gfCNCPoint2[25191] = {X 190.9402, Y 34.0721, Z -3.8333, A 0.000, B 0.000, C 0.000 }
gfCNCPoint2[25192] = {X 189.2026, Y 34.2446, Z -3.8333, A 0.000, B 0.000, C 0.000 }
gfCNCPoint2[25193] = {X 186.9380, Y 34.3837, Z -3.8333, A 0.000, B 0.000, C 0.000 }
gfCNCPoint2[25194] = {X 182.9821, Y 34.9758, Z -3.8333, A 0.000, B 0.000, C 0.000 }
gfCNCPoint2[25195] = {X 182.9821, Y 34.9758, Z -0.8333, A 0.000, B 0.000, C 0.000 }
gfCNCPoint2[25196] = {X 182.9821, Y 34.9758, Z 11.0000, A 0.000, B 0.000, C 0.000 }
gfCNCPoint2[25197] = {X 188.4961, Y 19.4662, Z 11.0000, A 0.000, B 0.000, C 0.000 }
gfCNCPoint2[25198] = {X 188.4961, Y 19.4662, Z 0.0000, A 0.000, B 0.000, C 0.000 }
gfCNCPoint2[25199] = {X 188.3884, Y 19.4281, Z -0.0306, A 0.000, B 0.000, C 0.000 }
gfCNCPoint2[25200] = {X 187.7714, Y 19.3596, Z -0.1969, A 0.000, B 0.000, C 0.000 }
gfCNCPoint2[25201] = {X 186.9109, Y 19.2596, Z -0.4291, A 0.000, B 0.000, C 0.000 }
gfCNCPoint2[25202] = {X 184.5930, Y 19.3671, Z -1.0508, A 0.000, B 0.000, C 0.000 }
gfCNCPoint2[25203] = {X 183.7430, Y 19.5468, Z -1.2836, A 0.000, B 0.000, C 0.000 }
gfCNCPoint2[25204] = {X 183.0416, Y 19.6905, Z -1.4754, A 0.000, B 0.000, C 0.000 }
gfCNCPoint2[25205] = {X 182.0251, Y 20.0604, Z -1.7653, A 0.000, B 0.000, C 0.000 }
gfCNCPoint2[25206] = {X 181.3955, Y 20.4012, Z -1.9571, A 0.000, B 0.000, C 0.000 }
gfCNCPoint2[25207] = {X 181.3396, Y 20.9128, Z -2.0950, A 0.000, B 0.000, C 0.000 }
gfCNCPoint2[25208] = {X 180.8645, Y 22.1268, Z -2.4443, A 0.000, B 0.000, C 0.000 }
gfCNCPoint2[25209] = {X 180.5584, Y 22.5405, Z -2.5822, A 0.000, B 0.000, C 0.000 }
gfCNCPoint2[25210] = {X 182.2910, Y 22.3346, Z -3.0498, A 0.000, B 0.000, C 0.000 }
gfCNCPoint2[25211] = {X 182.5945, Y 22.3099, Z -3.1314, A 0.000, B 0.000, C 0.000 }
gfCNCPoint2[25212] = {X 184.3413, Y 22.2338, Z -3.5999, A 0.000, B 0.000, C 0.000 }
gfCNCPoint2[25213] = {X 184.7767, Y 22.2187, Z -3.7166, A 0.000, B 0.000, C 0.000 }
gfCNCPoint2[25214] = {X 185.2120, Y 22.2003, Z -3.8333, A 0.000, B 0.000, C 0.000 }
gfCNCPoint2[25215] = {X 187.5425, Y 22.0778, Z -3.8333, A 0.000, B 0.000, C 0.000 }
gfCNCPoint2[25216] = {X 189.8700, Y 21.9074, Z -3.8333, A 0.000, B 0.000, C 0.000 }
gfCNCPoint2[25217] = {X 190.4716, Y 21.8313, Z -3.8333, A 0.000, B 0.000, C 0.000 }
gfCNCPoint2[25218] = {X 191.0588, Y 21.6799, Z -3.8333, A 0.000, B 0.000, C 0.000 }
gfCNCPoint2[25219] = {X 191.0686, Y 21.1639, Z -3.8333, A 0.000, B 0.000, C 0.000 }
gfCNCPoint2[25220] = {X 190.8728, Y 20.6864, Z -3.8333, A 0.000, B 0.000, C 0.000 }
gfCNCPoint2[25221] = {X 190.5036, Y 20.3258, Z -3.8333, A 0.000, B 0.000, C 0.000 }
gfCNCPoint2[25222] = {X 189.6459, Y 19.8651, Z -3.8333, A 0.000, B 0.000, C 0.000 }
gfCNCPoint2[25223] = {X 188.7281, Y 19.5404, Z -3.8333, A 0.000, B 0.000, C 0.000 }
gfCNCPoint2[25224] = {X 187.7714, Y 19.3596, Z -3.8333, A 0.000, B 0.000, C 0.000 }
gfCNCPoint2[25225] = {X 186.4245, Y 19.2765, Z -3.8333, A 0.000, B 0.000, C 0.000 }
gfCNCPoint2[25226] = {X 185.0764, Y 19.3391, Z -3.8333, A 0.000, B 0.000, C 0.000 }
gfCNCPoint2[25227] = {X 183.7430, Y 19.5468, Z -3.8333, A 0.000, B 0.000, C 0.000 }
gfCNCPoint2[25228] = {X 182.5378, Y 19.8876, Z -3.8333, A 0.000, B 0.000, C 0.000 }
gfCNCPoint2[25229] = {X 181.3955, Y 20.4012, Z -3.8333, A 0.000, B 0.000, C 0.000 }
gfCNCPoint2[25230] = {X 181.2441, Y 21.1600, Z -3.8333, A 0.000, B 0.000, C 0.000 }
gfCNCPoint2[25231] = {X 180.9622, Y 21.8805, Z -3.8333, A 0.000, B 0.000, C 0.000 }
gfCNCPoint2[25232] = {X 180.5584, Y 22.5405, Z -3.8333, A 0.000, B 0.000, C 0.000 }
gfCNCPoint2[25233] = {X 182.4470, Y 22.3518, Z -3.8333, A 0.000, B 0.000, C 0.000 }
gfCNCPoint2[25234] = {X 184.3413, Y 22.2338, Z -3.8333, A 0.000, B 0.000, C 0.000 }
gfCNCPoint2[25235] = {X 184.7767, Y 22.2179, Z -3.8333, A 0.000, B 0.000, C 0.000 }
gfCNCPoint2[25236] = {X 185.2120, Y 22.2003, Z -3.8333, A 0.000, B 0.000, C 0.000 }
gfCNCPoint2[25237] = {X 181.2194, Y 22.1003, Z -3.8333, A 0.000, B 0.000, C 0.000 }
gfCNCPoint2[25238] = {X 185.2154, Y 22.2803, Z -3.8333, A 0.000, B 0.000, C 0.000 }
gfCNCPoint2[25239] = {X 187.5451, Y 22.1578, Z -3.8333, A 0.000, B 0.000, C 0.000 }
gfCNCPoint2[25240] = {X 189.8718, Y 21.9874, Z -3.8333, A 0.000, B 0.000, C 0.000 }
gfCNCPoint2[25241] = {X 190.5070, Y 21.9059, Z -3.8333, A 0.000, B 0.000, C 0.000 }
gfCNCPoint2[25242] = {X 191.1260, Y 21.7420, Z -3.8333, A 0.000, B 0.000, C 0.000 }
gfCNCPoint2[25243] = {X 191.1525, Y 21.1792, Z -3.8333, A 0.000, B 0.000, C 0.000 }
gfCNCPoint2[25244] = {X 190.9475, Y 20.6544, Z -3.8333, A 0.000, B 0.000, C 0.000 }
gfCNCPoint2[25245] = {X 190.5467, Y 20.2585, Z -3.8333, A 0.000, B 0.000, C 0.000 }
gfCNCPoint2[25246] = {X 189.6789, Y 19.7922, Z -3.8333, A 0.000, B 0.000, C 0.000 }
gfCNCPoint2[25247] = {X 188.7502, Y 19.4636, Z -3.8333, A 0.000, B 0.000, C 0.000 }
gfCNCPoint2[25248] = {X 187.7823, Y 19.2803, Z -3.8333, A 0.000, B 0.000, C 0.000 }
gfCNCPoint2[25249] = {X 186.4270, Y 19.1965, Z -3.8333, A 0.000, B 0.000, C 0.000 }
gfCNCPoint2[25250] = {X 185.0706, Y 19.2593, Z -3.8333, A 0.000, B 0.000, C 0.000 }
gfCNCPoint2[25251] = {X 183.7289, Y 19.4680, Z -3.8333, A 0.000, B 0.000, C 0.000 }
gfCNCPoint2[25252] = {X 182.4922, Y 19.8190, Z -3.8333, A 0.000, B 0.000, C 0.000 }
gfCNCPoint2[25253] = {X 181.3215, Y 20.3504, Z -3.8333, A 0.000, B 0.000, C 0.000 }
gfCNCPoint2[25254] = {X 181.1595, Y 21.1706, Z -3.8333, A 0.000, B 0.000, C 0.000 }
gfCNCPoint2[25255] = {X 180.8425, Y 21.9443, Z -3.8333, A 0.000, B 0.000, C 0.000 }
gfCNCPoint2[25256] = {X 180.3824, Y 22.6424, Z -3.8333, A 0.000, B 0.000, C 0.000 }
gfCNCPoint2[25257] = {X 182.3593, Y 22.4392, Z -3.8333, A 0.000, B 0.000, C 0.000 }
gfCNCPoint2[25258] = {X 184.3427, Y 22.3138, Z -3.8333, A 0.000, B 0.000, C 0.000 }
gfCNCPoint2[25259] = {X 184.7791, Y 22.2979, Z -3.8333, A 0.000, B 0.000, C 0.000 }
gfCNCPoint2[25260] = {X 185.2154, Y 22.2803, Z -3.8333, A 0.000, B 0.000, C 0.000 }
gfCNCPoint2[25261] = {X 189.1819, Y 21.7636, Z -3.8333, A 0.000, B 0.000, C 0.000 }
gfCNCPoint2[25262] = {X 181.2228, Y 22.1802, Z -3.8333, A 0.000, B 0.000, C 0.000 }
gfCNCPoint2[25263] = {X 185.2187, Y 22.3602, Z -3.8333, A 0.000, B 0.000, C 0.000 }
gfCNCPoint2[25264] = {X 187.5497, Y 22.2376, Z -3.8333, A 0.000, B 0.000, C 0.000 }
gfCNCPoint2[25265] = {X 189.8776, Y 22.0672, Z -3.8333, A 0.000, B 0.000, C 0.000 }
gfCNCPoint2[25266] = {X 190.5436, Y 21.9802, Z -3.8333, A 0.000, B 0.000, C 0.000 }
gfCNCPoint2[25267] = {X 191.1918, Y 21.8041, Z -3.8333, A 0.000, B 0.000, C 0.000 }
gfCNCPoint2[25268] = {X 191.2495, Y 21.3480, Z -3.8333, A 0.000, B 0.000, C 0.000 }
gfCNCPoint2[25269] = {X 191.1599, Y 20.8972, Z -3.8333, A 0.000, B 0.000, C 0.000 }
gfCNCPoint2[25270] = {X 190.9322, Y 20.4978, Z -3.8333, A 0.000, B 0.000, C 0.000 }
gfCNCPoint2[25271] = {X 190.5898, Y 20.1911, Z -3.8333, A 0.000, B 0.000, C 0.000 }
gfCNCPoint2[25272] = {X 189.7113, Y 19.7190, Z -3.8333, A 0.000, B 0.000, C 0.000 }
gfCNCPoint2[25273] = {X 188.7710, Y 19.3863, Z -3.8333, A 0.000, B 0.000, C 0.000 }
gfCNCPoint2[25274] = {X 187.7911, Y 19.2008, Z -3.8333, A 0.000, B 0.000, C 0.000 }
gfCNCPoint2[25275] = {X 186.4273, Y 19.1165, Z -3.8333, A 0.000, B 0.000, C 0.000 }
gfCNCPoint2[25276] = {X 185.0625, Y 19.1797, Z -3.8333, A 0.000, B 0.000, C 0.000 }
gfCNCPoint2[25277] = {X 183.7123, Y 19.3897, Z -3.8333, A 0.000, B 0.000, C 0.000 }
gfCNCPoint2[25278] = {X 182.4466, Y 19.7506, Z -3.8333, A 0.000, B 0.000, C 0.000 }
gfCNCPoint2[25279] = {X 181.2499, Y 20.2985, Z -3.8333, A 0.000, B 0.000, C 0.000 }
gfCNCPoint2[25280] = {X 181.2398, Y 20.3524, Z -3.8333, A 0.000, B 0.000, C 0.000 }
gfCNCPoint2[25281] = {X 181.0601, Y 21.2185, Z -3.8333, A 0.000, B 0.000, C 0.000 }
gfCNCPoint2[25282] = {X 180.7046, Y 22.0285, Z -3.8333, A 0.000, B 0.000, C 0.000 }
gfCNCPoint2[25283] = {X 180.1888, Y 22.7471, Z -3.8333, A 0.000, B 0.000, C 0.000 }
gfCNCPoint2[25284] = {X 182.2636, Y 22.5276, Z -3.8333, A 0.000, B 0.000, C 0.000 }
gfCNCPoint2[25285] = {X 184.3458, Y 22.3938, Z -3.8333, A 0.000, B 0.000, C 0.000 }
gfCNCPoint2[25286] = {X 184.7823, Y 22.3778, Z -3.8333, A 0.000, B 0.000, C 0.000 }
gfCNCPoint2[25287] = {X 185.2187, Y 22.3602, Z -3.8333, A 0.000, B 0.000, C 0.000 }
gfCNCPoint2[25288] = {X 189.1852, Y 21.8435, Z -3.8333, A 0.000, B 0.000, C 0.000 }
gfCNCPoint2[25289] = {X 181.2262, Y 22.2602, Z -3.8333, A 0.000, B 0.000, C 0.000 }
gfCNCPoint2[25290] = {X 185.2221, Y 22.4401, Z -3.8333, A 0.000, B 0.000, C 0.000 }
gfCNCPoint2[25291] = {X 187.5543, Y 22.3175, Z -3.8333, A 0.000, B 0.000, C 0.000 }
gfCNCPoint2[25292] = {X 189.8834, Y 22.1470, Z -3.8333, A 0.000, B 0.000, C 0.000 }
gfCNCPoint2[25293] = {X 190.5796, Y 22.0546, Z -3.8333, A 0.000, B 0.000, C 0.000 }
gfCNCPoint2[25294] = {X 191.2562, Y 21.8662, Z -3.8333, A 0.000, B 0.000, C 0.000 }
gfCNCPoint2[25295] = {X 191.3302, Y 21.3762, Z -3.8333, A 0.000, B 0.000, C 0.000 }
gfCNCPoint2[25296] = {X 191.2419, Y 20.8886, Z -3.8333, A 0.000, B 0.000, C 0.000 }
gfCNCPoint2[25297] = {X 191.0009, Y 20.4557, Z -3.8333, A 0.000, B 0.000, C 0.000 }
gfCNCPoint2[25298] = {X 190.6330, Y 20.1237, Z -3.8333, A 0.000, B 0.000, C 0.000 }
gfCNCPoint2[25299] = {X 189.7437, Y 19.6459, Z -3.8333, A 0.000, B 0.000, C 0.000 }
gfCNCPoint2[25300] = {X 188.7919, Y 19.3091, Z -3.8333, A 0.000, B 0.000, C 0.000 }
gfCNCPoint2[25301] = {X 187.7999, Y 19.1213, Z -3.8333, A 0.000, B 0.000, C 0.000 }
gfCNCPoint2[25302] = {X 186.4277, Y 19.0365, Z -3.8333, A 0.000, B 0.000, C 0.000 }
gfCNCPoint2[25303] = {X 185.0543, Y 19.1001, Z -3.8333, A 0.000, B 0.000, C 0.000 }
gfCNCPoint2[25304] = {X 183.6958, Y 19.3115, Z -3.8333, A 0.000, B 0.000, C 0.000 }
gfCNCPoint2[25305] = {X 182.4009, Y 19.6822, Z -3.8333, A 0.000, B 0.000, C 0.000 }
gfCNCPoint2[25306] = {X 181.1781, Y 20.2468, Z -3.8333, A 0.000, B 0.000, C 0.000 }
gfCNCPoint2[25307] = {X 181.1605, Y 20.3410, Z -3.8333, A 0.000, B 0.000, C 0.000 }
gfCNCPoint2[25308] = {X 180.9651, Y 21.2476, Z -3.8333, A 0.000, B 0.000, C 0.000 }
gfCNCPoint2[25309] = {X 180.5736, Y 22.0884, Z -3.8333, A 0.000, B 0.000, C 0.000 }
gfCNCPoint2[25310] = {X 180.0056, Y 22.8216, Z -3.8333, A 0.000, B 0.000, C 0.000 }
gfCNCPoint2[25311] = {X 180.1926, Y 22.8273, Z -3.8333, A 0.000, B 0.000, C 0.000 }
gfCNCPoint2[25312] = {X 182.2671, Y 22.6075, Z -3.8333, A 0.000, B 0.000, C 0.000 }
gfCNCPoint2[25313] = {X 184.3489, Y 22.4737, Z -3.8333, A 0.000, B 0.000, C 0.000 }
gfCNCPoint2[25314] = {X 184.7856, Y 22.4577, Z -3.8333, A 0.000, B 0.000, C 0.000 }
gfCNCPoint2[25315] = {X 185.2221, Y 22.4401, Z -3.8333, A 0.000, B 0.000, C 0.000 }
gfCNCPoint2[25316] = {X 189.1886, Y 21.9235, Z -3.8333, A 0.000, B 0.000, C 0.000 }
gfCNCPoint2[25317] = {X 181.2296, Y 22.3401, Z -3.8333, A 0.000, B 0.000, C 0.000 }
gfCNCPoint2[25318] = {X 185.2255, Y 22.5201, Z -3.8333, A 0.000, B 0.000, C 0.000 }
gfCNCPoint2[25319] = {X 187.5589, Y 22.3974, Z -3.8333, A 0.000, B 0.000, C 0.000 }
gfCNCPoint2[25320] = {X 189.8892, Y 22.2268, Z -3.8333, A 0.000, B 0.000, C 0.000 }
gfCNCPoint2[25321] = {X 190.6151, Y 22.1289, Z -3.8333, A 0.000, B 0.000, C 0.000 }
gfCNCPoint2[25322] = {X 191.3196, Y 21.9285, Z -3.8333, A 0.000, B 0.000, C 0.000 }
gfCNCPoint2[25323] = {X 191.4103, Y 21.4048, Z -3.8333, A 0.000, B 0.000, C 0.000 }
gfCNCPoint2[25324] = {X 191.3238, Y 20.8804, Z -3.8333, A 0.000, B 0.000, C 0.000 }
gfCNCPoint2[25325] = {X 191.0696, Y 20.4136, Z -3.8333, A 0.000, B 0.000, C 0.000 }
gfCNCPoint2[25326] = {X 190.6761, Y 20.0564, Z -3.8333, A 0.000, B 0.000, C 0.000 }
gfCNCPoint2[25327] = {X 189.7760, Y 19.5727, Z -3.8333, A 0.000, B 0.000, C 0.000 }
gfCNCPoint2[25328] = {X 188.8127, Y 19.2318, Z -3.8333, A 0.000, B 0.000, C 0.000 }
gfCNCPoint2[25329] = {X 187.8088, Y 19.0418, Z -3.8333, A 0.000, B 0.000, C 0.000 }
gfCNCPoint2[25330] = {X 186.4280, Y 18.9565, Z -3.8333, A 0.000, B 0.000, C 0.000 }
gfCNCPoint2[25331] = {X 185.0462, Y 19.0205, Z -3.8333, A 0.000, B 0.000, C 0.000 }
gfCNCPoint2[25332] = {X 183.6792, Y 19.2332, Z -3.8333, A 0.000, B 0.000, C 0.000 }
gfCNCPoint2[25333] = {X 182.3552, Y 19.6138, Z -3.8333, A 0.000, B 0.000, C 0.000 }
gfCNCPoint2[25334] = {X 181.1064, Y 20.1954, Z -3.8333, A 0.000, B 0.000, C 0.000 }
gfCNCPoint2[25335] = {X 181.0813, Y 20.3296, Z -3.8333, A 0.000, B 0.000, C 0.000 }
gfCNCPoint2[25336] = {X 180.8699, Y 21.2784, Z -3.8333, A 0.000, B 0.000, C 0.000 }
gfCNCPoint2[25337] = {X 180.4400, Y 22.1503, Z -3.8333, A 0.000, B 0.000, C 0.000 }
gfCNCPoint2[25338] = {X 179.8161, Y 22.8958, Z -3.8333, A 0.000, B 0.000, C 0.000 }
gfCNCPoint2[25339] = {X 180.1964, Y 22.9074, Z -3.8333, A 0.000, B 0.000, C 0.000 }
gfCNCPoint2[25340] = {X 182.2706, Y 22.6875, Z -3.8333, A 0.000, B 0.000, C 0.000 }
gfCNCPoint2[25341] = {X 184.3521, Y 22.5536, Z -3.8333, A 0.000, B 0.000, C 0.000 }
gfCNCPoint2[25342] = {X 184.7888, Y 22.5377, Z -3.8333, A 0.000, B 0.000, C 0.000 }
gfCNCPoint2[25343] = {X 185.2255, Y 22.5201, Z -3.8333, A 0.000, B 0.000, C 0.000 }
gfCNCPoint2[25344] = {X 189.1920, Y 22.0034, Z -3.8333, A 0.000, B 0.000, C 0.000 }
gfCNCPoint2[25345] = {X 185.1538, Y 22.6031, Z -3.8333, A 0.000, B 0.000, C 0.000 }
gfCNCPoint2[25346] = {X 185.2289, Y 22.6000, Z -3.8333, A 0.000, B 0.000, C 0.000 }
gfCNCPoint2[25347] = {X 187.5635, Y 22.4772, Z -3.8333, A 0.000, B 0.000, C 0.000 }
gfCNCPoint2[25348] = {X 189.8950, Y 22.3066, Z -3.8333, A 0.000, B 0.000, C 0.000 }
gfCNCPoint2[25349] = {X 190.6501, Y 22.2033, Z -3.8333, A 0.000, B 0.000, C 0.000 }
gfCNCPoint2[25350] = {X 191.3820, Y 21.9907, Z -3.8333, A 0.000, B 0.000, C 0.000 }
gfCNCPoint2[25351] = {X 191.4900, Y 21.4336, Z -3.8333, A 0.000, B 0.000, C 0.000 }
gfCNCPoint2[25352] = {X 191.4055, Y 20.8724, Z -3.8333, A 0.000, B 0.000, C 0.000 }
gfCNCPoint2[25353] = {X 191.1384, Y 20.3716, Z -3.8333, A 0.000, B 0.000, C 0.000 }
gfCNCPoint2[25354] = {X 190.7193, Y 19.9890, Z -3.8333, A 0.000, B 0.000, C 0.000 }
gfCNCPoint2[25355] = {X 189.8084, Y 19.4995, Z -3.8333, A 0.000, B 0.000, C 0.000 }
gfCNCPoint2[25356] = {X 188.8336, Y 19.1546, Z -3.8333, A 0.000, B 0.000, C 0.000 }
gfCNCPoint2[25357] = {X 187.8176, Y 18.9622, Z -3.8333, A 0.000, B 0.000, C 0.000 }
gfCNCPoint2[25358] = {X 186.4284, Y 18.8765, Z -3.8333, A 0.000, B 0.000, C 0.000 }
gfCNCPoint2[25359] = {X 185.0380, Y 18.9410, Z -3.8333, A 0.000, B 0.000, C 0.000 }
gfCNCPoint2[25360] = {X 183.6627, Y 19.1549, Z -3.8333, A 0.000, B 0.000, C 0.000 }
gfCNCPoint2[25361] = {X 182.3095, Y 19.5455, Z -3.8333, A 0.000, B 0.000, C 0.000 }
gfCNCPoint2[25362] = {X 181.0346, Y 20.1441, Z -3.8333, A 0.000, B 0.000, C 0.000 }
gfCNCPoint2[25363] = {X 181.0020, Y 20.3183, Z -3.8333, A 0.000, B 0.000, C 0.000 }
gfCNCPoint2[25364] = {X 180.8538, Y 21.0695, Z -3.8333, A 0.000, B 0.000, C 0.000 }
gfCNCPoint2[25365] = {X 180.5651, Y 21.7787, Z -3.8333, A 0.000, B 0.000, C 0.000 }
gfCNCPoint2[25366] = {X 180.1466, Y 22.4199, Z -3.8333, A 0.000, B 0.000, C 0.000 }
gfCNCPoint2[25367] = {X 179.6136, Y 22.9696, Z -3.8333, A 0.000, B 0.000, C 0.000 }
gfCNCPoint2[25368] = {X 180.2003, Y 22.9876, Z -3.8333, A 0.000, B 0.000, C 0.000 }
gfCNCPoint2[25369] = {X 182.2741, Y 22.7675, Z -3.8333, A 0.000, B 0.000, C 0.000 }
gfCNCPoint2[25370] = {X 184.3552, Y 22.6336, Z -3.8333, A 0.000, B 0.000, C 0.000 }
gfCNCPoint2[25371] = {X 184.7921, Y 22.6176, Z -3.8333, A 0.000, B 0.000, C 0.000 }
gfCNCPoint2[25372] = {X 185.2289, Y 22.6000, Z -3.8333, A 0.000, B 0.000, C 0.000 }
gfCNCPoint2[25373] = {X 185.1444, Y 20.6018, Z -3.8333, A 0.000, B 0.000, C 0.000 }
gfCNCPoint2[25374] = {X 185.1444, Y 20.6018, Z -0.8333, A 0.000, B 0.000, C 0.000 }
gfCNCPoint2[25375] = {X 185.1444, Y 20.6018, Z 11.0000, A 0.000, B 0.000, C 0.000 }
gfCNCPoint2[25376] = {X 256.2436, Y 19.7807, Z 11.0000, A 0.000, B 0.000, C 0.000 }
gfCNCPoint2[25377] = {X 256.2436, Y 19.7807, Z 0.0000, A 0.000, B 0.000, C 0.000 }
gfCNCPoint2[25378] = {X 251.5292, Y 19.7807, Z -1.2632, A 0.000, B 0.000, C 0.000 }
gfCNCPoint2[25379] = {X 250.8345, Y 19.7916, Z -1.4494, A 0.000, B 0.000, C 0.000 }
gfCNCPoint2[25380] = {X 250.1809, Y 19.7930, Z -1.6245, A 0.000, B 0.000, C 0.000 }
gfCNCPoint2[25381] = {X 249.4954, Y 19.8914, Z -1.8101, A 0.000, B 0.000, C 0.000 }
gfCNCPoint2[25382] = {X 248.8452, Y 20.0797, Z -1.9915, A 0.000, B 0.000, C 0.000 }
gfCNCPoint2[25383] = {X 248.7082, Y 20.1110, Z -2.0291, A 0.000, B 0.000, C 0.000 }
gfCNCPoint2[25384] = {X 248.6540, Y 20.1618, Z -2.0490, A 0.000, B 0.000, C 0.000 }
gfCNCPoint2[25385] = {X 248.4750, Y 20.7647, Z -2.2175, A 0.000, B 0.000, C 0.000 }
gfCNCPoint2[25386] = {X 248.4449, Y 21.8677, Z -2.5132, A 0.000, B 0.000, C 0.000 }
gfCNCPoint2[25387] = {X 248.5581, Y 22.3427, Z -2.6441, A 0.000, B 0.000, C 0.000 }
gfCNCPoint2[25388] = {X 248.8730, Y 22.4374, Z -2.7322, A 0.000, B 0.000, C 0.000 }
gfCNCPoint2[25389] = {X 249.2007, Y 22.4646, Z -2.8203, A 0.000, B 0.000, C 0.000 }
gfCNCPoint2[25390] = {X 250.4401, Y 22.5675, Z -3.1535, A 0.000, B 0.000, C 0.000 }
gfCNCPoint2[25391] = {X 251.6873, Y 22.5560, Z -3.4877, A 0.000, B 0.000, C 0.000 }
gfCNCPoint2[25392] = {X 252.9772, Y 22.5560, Z -3.8333, A 0.000, B 0.000, C 0.000 }
gfCNCPoint2[25393] = {X 257.4115, Y 22.5560, Z -3.8333, A 0.000, B 0.000, C 0.000 }
gfCNCPoint2[25394] = {X 257.4115, Y 19.7807, Z -3.8333, A 0.000, B 0.000, C 0.000 }
gfCNCPoint2[25395] = {X 251.5292, Y 19.7807, Z -3.8333, A 0.000, B 0.000, C 0.000 }
gfCNCPoint2[25396] = {X 250.8345, Y 19.7916, Z -3.8333, A 0.000, B 0.000, C 0.000 }
gfCNCPoint2[25397] = {X 249.8296, Y 19.8649, Z -3.8333, A 0.000, B 0.000, C 0.000 }
gfCNCPoint2[25398] = {X 248.8452, Y 20.0797, Z -3.8333, A 0.000, B 0.000, C 0.000 }
gfCNCPoint2[25399] = {X 248.7002, Y 20.1568, Z -3.8333, A 0.000, B 0.000, C 0.000 }
gfCNCPoint2[25400] = {X 248.6140, Y 20.2965, Z -3.8333, A 0.000, B 0.000, C 0.000 }
gfCNCPoint2[25401] = {X 248.4760, Y 20.9719, Z -3.8333, A 0.000, B 0.000, C 0.000 }
gfCNCPoint2[25402] = {X 248.4572, Y 21.6609, Z -3.8333, A 0.000, B 0.000, C 0.000 }
gfCNCPoint2[25403] = {X 248.5581, Y 22.3427, Z -3.8333, A 0.000, B 0.000, C 0.000 }
gfCNCPoint2[25404] = {X 248.8762, Y 22.4205, Z -3.8333, A 0.000, B 0.000, C 0.000 }
gfCNCPoint2[25405] = {X 249.2007, Y 22.4646, Z -3.8333, A 0.000, B 0.000, C 0.000 }
gfCNCPoint2[25406] = {X 250.4430, Y 22.5389, Z -3.8333, A 0.000, B 0.000, C 0.000 }
gfCNCPoint2[25407] = {X 251.6873, Y 22.5560, Z -3.8333, A 0.000, B 0.000, C 0.000 }
gfCNCPoint2[25408] = {X 252.9772, Y 22.5560, Z -3.8333, A 0.000, B 0.000, C 0.000 }
gfCNCPoint2[25409] = {X 248.9925, Y 22.2874, Z -3.8333, A 0.000, B 0.000, C 0.000 }
gfCNCPoint2[25410] = {X 252.9772, Y 22.6360, Z -3.8333, A 0.000, B 0.000, C 0.000 }
gfCNCPoint2[25411] = {X 257.4915, Y 22.6360, Z -3.8333, A 0.000, B 0.000, C 0.000 }
gfCNCPoint2[25412] = {X 257.4915, Y 19.7007, Z -3.8333, A 0.000, B 0.000, C 0.000 }
gfCNCPoint2[25413] = {X 251.5286, Y 19.7007, Z -3.8333, A 0.000, B 0.000, C 0.000 }
gfCNCPoint2[25414] = {X 250.8365, Y 19.7116, Z -3.8333, A 0.000, B 0.000, C 0.000 }
gfCNCPoint2[25415] = {X 249.8259, Y 19.7850, Z -3.8333, A 0.000, B 0.000, C 0.000 }
gfCNCPoint2[25416] = {X 248.8356, Y 19.9999, Z -3.8333, A 0.000, B 0.000, C 0.000 }
gfCNCPoint2[25417] = {X 248.6486, Y 20.0956, Z -3.8333, A 0.000, B 0.000, C 0.000 }
gfCNCPoint2[25418] = {X 248.5373, Y 20.2738, Z -3.8333, A 0.000, B 0.000, C 0.000 }
gfCNCPoint2[25419] = {X 248.3948, Y 20.9779, Z -3.8333, A 0.000, B 0.000, C 0.000 }
gfCNCPoint2[25420] = {X 248.3793, Y 21.6962, Z -3.8333, A 0.000, B 0.000, C 0.000 }
gfCNCPoint2[25421] = {X 248.4912, Y 22.4058, Z -3.8333, A 0.000, B 0.000, C 0.000 }
gfCNCPoint2[25422] = {X 248.8388, Y 22.4947, Z -3.8333, A 0.000, B 0.000, C 0.000 }
gfCNCPoint2[25423] = {X 249.1941, Y 22.5443, Z -3.8333, A 0.000, B 0.000, C 0.000 }
gfCNCPoint2[25424] = {X 250.4389, Y 22.6188, Z -3.8333, A 0.000, B 0.000, C 0.000 }
gfCNCPoint2[25425] = {X 251.6859, Y 22.6360, Z -3.8333, A 0.000, B 0.000, C 0.000 }
gfCNCPoint2[25426] = {X 252.9772, Y 22.6360, Z -3.8333, A 0.000, B 0.000, C 0.000 }
gfCNCPoint2[25427] = {X 256.9620, Y 22.2874, Z -3.8333, A 0.000, B 0.000, C 0.000 }
gfCNCPoint2[25428] = {X 248.9925, Y 22.3674, Z -3.8333, A 0.000, B 0.000, C 0.000 }
gfCNCPoint2[25429] = {X 252.9772, Y 22.7160, Z -3.8333, A 0.000, B 0.000, C 0.000 }
gfCNCPoint2[25430] = {X 257.5715, Y 22.7160, Z -3.8333, A 0.000, B 0.000, C 0.000 }
gfCNCPoint2[25431] = {X 257.5715, Y 19.6207, Z -3.8333, A 0.000, B 0.000, C 0.000 }
gfCNCPoint2[25432] = {X 251.5280, Y 19.6207, Z -3.8333, A 0.000, B 0.000, C 0.000 }
gfCNCPoint2[25433] = {X 250.8358, Y 19.6316, Z -3.8333, A 0.000, B 0.000, C 0.000 }
gfCNCPoint2[25434] = {X 249.8156, Y 19.7056, Z -3.8333, A 0.000, B 0.000, C 0.000 }
gfCNCPoint2[25435] = {X 248.8160, Y 19.9223, Z -3.8333, A 0.000, B 0.000, C 0.000 }
gfCNCPoint2[25436] = {X 248.5932, Y 20.0379, Z -3.8333, A 0.000, B 0.000, C 0.000 }
gfCNCPoint2[25437] = {X 248.4606, Y 20.2510, Z -3.8333, A 0.000, B 0.000, C 0.000 }
gfCNCPoint2[25438] = {X 248.3137, Y 20.9838, Z -3.8333, A 0.000, B 0.000, C 0.000 }
gfCNCPoint2[25439] = {X 248.3016, Y 21.7311, Z -3.8333, A 0.000, B 0.000, C 0.000 }
gfCNCPoint2[25440] = {X 248.4247, Y 22.4684, Z -3.8333, A 0.000, B 0.000, C 0.000 }
gfCNCPoint2[25441] = {X 248.8014, Y 22.5688, Z -3.8333, A 0.000, B 0.000, C 0.000 }
gfCNCPoint2[25442] = {X 249.1874, Y 22.6240, Z -3.8333, A 0.000, B 0.000, C 0.000 }
gfCNCPoint2[25443] = {X 250.4358, Y 22.6988, Z -3.8333, A 0.000, B 0.000, C 0.000 }
gfCNCPoint2[25444] = {X 251.6862, Y 22.7160, Z -3.8333, A 0.000, B 0.000, C 0.000 }
gfCNCPoint2[25445] = {X 252.9772, Y 22.7160, Z -3.8333, A 0.000, B 0.000, C 0.000 }
gfCNCPoint2[25446] = {X 256.9620, Y 22.3674, Z -3.8333, A 0.000, B 0.000, C 0.000 }
gfCNCPoint2[25447] = {X 248.9925, Y 22.4474, Z -3.8333, A 0.000, B 0.000, C 0.000 }
gfCNCPoint2[25448] = {X 252.9772, Y 22.7960, Z -3.8333, A 0.000, B 0.000, C 0.000 }
gfCNCPoint2[25449] = {X 257.6515, Y 22.7960, Z -3.8333, A 0.000, B 0.000, C 0.000 }
gfCNCPoint2[25450] = {X 257.6515, Y 19.5407, Z -3.8333, A 0.000, B 0.000, C 0.000 }
gfCNCPoint2[25451] = {X 251.5274, Y 19.5407, Z -3.8333, A 0.000, B 0.000, C 0.000 }
gfCNCPoint2[25452] = {X 250.8351, Y 19.5516, Z -3.8333, A 0.000, B 0.000, C 0.000 }
gfCNCPoint2[25453] = {X 249.8053, Y 19.6263, Z -3.8333, A 0.000, B 0.000, C 0.000 }
gfCNCPoint2[25454] = {X 248.7962, Y 19.8447, Z -3.8333, A 0.000, B 0.000, C 0.000 }
gfCNCPoint2[25455] = {X 248.5377, Y 19.9802, Z -3.8333, A 0.000, B 0.000, C 0.000 }
gfCNCPoint2[25456] = {X 248.3839, Y 20.2282, Z -3.8333, A 0.000, B 0.000, C 0.000 }
gfCNCPoint2[25457] = {X 248.2326, Y 20.9896, Z -3.8333, A 0.000, B 0.000, C 0.000 }
gfCNCPoint2[25458] = {X 248.2241, Y 21.7659, Z -3.8333, A 0.000, B 0.000, C 0.000 }
gfCNCPoint2[25459] = {X 248.3584, Y 22.5304, Z -3.8333, A 0.000, B 0.000, C 0.000 }
gfCNCPoint2[25460] = {X 248.7642, Y 22.6428, Z -3.8333, A 0.000, B 0.000, C 0.000 }
gfCNCPoint2[25461] = {X 249.1808, Y 22.7037, Z -3.8333, A 0.000, B 0.000, C 0.000 }
gfCNCPoint2[25462] = {X 250.4327, Y 22.7787, Z -3.8333, A 0.000, B 0.000, C 0.000 }
gfCNCPoint2[25463] = {X 251.6866, Y 22.7960, Z -3.8333, A 0.000, B 0.000, C 0.000 }
gfCNCPoint2[25464] = {X 252.9772, Y 22.7960, Z -3.8333, A 0.000, B 0.000, C 0.000 }
gfCNCPoint2[25465] = {X 256.9620, Y 22.4474, Z -3.8333, A 0.000, B 0.000, C 0.000 }
gfCNCPoint2[25466] = {X 248.9925, Y 22.5274, Z -3.8333, A 0.000, B 0.000, C 0.000 }
gfCNCPoint2[25467] = {X 252.9772, Y 22.8760, Z -3.8333, A 0.000, B 0.000, C 0.000 }
gfCNCPoint2[25468] = {X 257.7315, Y 22.8760, Z -3.8333, A 0.000, B 0.000, C 0.000 }
gfCNCPoint2[25469] = {X 257.7315, Y 19.4607, Z -3.8333, A 0.000, B 0.000, C 0.000 }
gfCNCPoint2[25470] = {X 251.5267, Y 19.4607, Z -3.8333, A 0.000, B 0.000, C 0.000 }
gfCNCPoint2[25471] = {X 250.8344, Y 19.4716, Z -3.8333, A 0.000, B 0.000, C 0.000 }
gfCNCPoint2[25472] = {X 249.7949, Y 19.5470, Z -3.8333, A 0.000, B 0.000, C 0.000 }
gfCNCPoint2[25473] = {X 248.7763, Y 19.7672, Z -3.8333, A 0.000, B 0.000, C 0.000 }
gfCNCPoint2[25474] = {X 248.4822, Y 19.9226, Z -3.8333, A 0.000, B 0.000, C 0.000 }
gfCNCPoint2[25475] = {X 248.3072, Y 20.2054, Z -3.8333, A 0.000, B 0.000, C 0.000 }
gfCNCPoint2[25476] = {X 248.1523, Y 20.9889, Z -3.8333, A 0.000, B 0.000, C 0.000 }
gfCNCPoint2[25477] = {X 248.1456, Y 21.7875, Z -3.8333, A 0.000, B 0.000, C 0.000 }
gfCNCPoint2[25478] = {X 248.2873, Y 22.5734, Z -3.8333, A 0.000, B 0.000, C 0.000 }
gfCNCPoint2[25479] = {X 248.3060, Y 22.5968, Z -3.8333, A 0.000, B 0.000, C 0.000 }
gfCNCPoint2[25480] = {X 248.3323, Y 22.6060, Z -3.8333, A 0.000, B 0.000, C 0.000 }
gfCNCPoint2[25481] = {X 248.7477, Y 22.7211, Z -3.8333, A 0.000, B 0.000, C 0.000 }
gfCNCPoint2[25482] = {X 249.1742, Y 22.7835, Z -3.8333, A 0.000, B 0.000, C 0.000 }
gfCNCPoint2[25483] = {X 250.4295, Y 22.8587, Z -3.8333, A 0.000, B 0.000, C 0.000 }
gfCNCPoint2[25484] = {X 251.6870, Y 22.8760, Z -3.8333, A 0.000, B 0.000, C 0.000 }
gfCNCPoint2[25485] = {X 252.9772, Y 22.8760, Z -3.8333, A 0.000, B 0.000, C 0.000 }
gfCNCPoint2[25486] = {X 256.9620, Y 22.5274, Z -3.8333, A 0.000, B 0.000, C 0.000 }
gfCNCPoint2[25487] = {X 252.9772, Y 20.9560, Z -3.8333, A 0.000, B 0.000, C 0.000 }
gfCNCPoint2[25488] = {X 252.9772, Y 22.9560, Z -3.8333, A 0.000, B 0.000, C 0.000 }
gfCNCPoint2[25489] = {X 257.8115, Y 22.9560, Z -3.8333, A 0.000, B 0.000, C 0.000 }
gfCNCPoint2[25490] = {X 257.8090, Y 19.3807, Z -3.8333, A 0.000, B 0.000, C 0.000 }
gfCNCPoint2[25491] = {X 251.5261, Y 19.3807, Z -3.8333, A 0.000, B 0.000, C 0.000 }
gfCNCPoint2[25492] = {X 250.8336, Y 19.3916, Z -3.8333, A 0.000, B 0.000, C 0.000 }
gfCNCPoint2[25493] = {X 249.7844, Y 19.4677, Z -3.8333, A 0.000, B 0.000, C 0.000 }
gfCNCPoint2[25494] = {X 248.7562, Y 19.6897, Z -3.8333, A 0.000, B 0.000, C 0.000 }
gfCNCPoint2[25495] = {X 248.4266, Y 19.8650, Z -3.8333, A 0.000, B 0.000, C 0.000 }
gfCNCPoint2[25496] = {X 248.2305, Y 20.1827, Z -3.8333, A 0.000, B 0.000, C 0.000 }
gfCNCPoint2[25497] = {X 248.0722, Y 20.9862, Z -3.8333, A 0.000, B 0.000, C 0.000 }
gfCNCPoint2[25498] = {X 248.0668, Y 21.8051, Z -3.8333, A 0.000, B 0.000, C 0.000 }
gfCNCPoint2[25499] = {X 248.2147, Y 22.6106, Z -3.8333, A 0.000, B 0.000, C 0.000 }
gfCNCPoint2[25500] = {X 248.2577, Y 22.6645, Z -3.8333, A 0.000, B 0.000, C 0.000 }
gfCNCPoint2[25501] = {X 248.7061, Y 22.7940, Z -3.8333, A 0.000, B 0.000, C 0.000 }
gfCNCPoint2[25502] = {X 249.1676, Y 22.8632, Z -3.8333, A 0.000, B 0.000, C 0.000 }
gfCNCPoint2[25503] = {X 250.4264, Y 22.9386, Z -3.8333, A 0.000, B 0.000, C 0.000 }
gfCNCPoint2[25504] = {X 251.6873, Y 22.9560, Z -3.8333, A 0.000, B 0.000, C 0.000 }
gfCNCPoint2[25505] = {X 252.9772, Y 22.9560, Z -3.8333, A 0.000, B 0.000, C 0.000 }
gfCNCPoint2[25506] = {X 256.9772, Y 22.9560, Z -3.8333, A 0.000, B 0.000, C 0.000 }
gfCNCPoint2[25507] = {X 256.9772, Y 22.9560, Z -0.8333, A 0.000, B 0.000, C 0.000 }
gfCNCPoint2[25508] = {X 256.9772, Y 22.9560, Z 11.0000, A 0.000, B 0.000, C 0.000 }
gfCNCPoint2[25509] = {X 507.6816, Y 107.6950, Z 11.0000, A 0.000, B 0.000, C 0.000 }
gfCNCPoint2[25510] = {X 507.6816, Y 107.6950, Z -0.8333, A 0.000, B 0.000, C 0.000 }
gfCNCPoint2[25511] = {X 507.6816, Y 107.6950, Z -3.8333, A 0.000, B 0.000, C 0.000 }
gfCNCPoint2[25512] = {X 507.6816, Y 71.2950, Z -3.8333, A 0.000, B 0.000, C 0.000 }
gfCNCPoint2[25513] = {X 509.5501, Y 71.2950, Z -3.8333, A 0.000, B 0.000, C 0.000 }
gfCNCPoint2[25514] = {X 509.0278, Y 71.0691, Z -3.8333, A 0.000, B 0.000, C 0.000 }
gfCNCPoint2[25515] = {X 508.5105, Y 70.8320, Z -3.8333, A 0.000, B 0.000, C 0.000 }
gfCNCPoint2[25516] = {X 507.1678, Y 71.0984, Z -3.8333, A 0.000, B 0.000, C 0.000 }
gfCNCPoint2[25517] = {X 505.8132, Y 71.2950, Z -3.8333, A 0.000, B 0.000, C 0.000 }
gfCNCPoint2[25518] = {X 507.6816, Y 71.2950, Z -3.8333, A 0.000, B 0.000, C 0.000 }
gfCNCPoint2[25519] = {X 507.6816, Y 73.6950, Z -3.8333, A 0.000, B 0.000, C 0.000 }
gfCNCPoint2[25520] = {X 551.2534, Y 73.6950, Z -3.8333, A 0.000, B 0.000, C 0.000 }
gfCNCPoint2[25521] = {X 549.1236, Y 72.7705, Z -3.8333, A 0.000, B 0.000, C 0.000 }
gfCNCPoint2[25522] = {X 547.0696, Y 71.6882, Z -3.8333, A 0.000, B 0.000, C 0.000 }
gfCNCPoint2[25523] = {X 545.1029, Y 70.4542, Z -3.8333, A 0.000, B 0.000, C 0.000 }
gfCNCPoint2[25524] = {X 543.2348, Y 69.0756, Z -3.8333, A 0.000, B 0.000, C 0.000 }
gfCNCPoint2[25525] = {X 529.7636, Y 69.0759, Z -3.8333, A 0.000, B 0.000, C 0.000 }
gfCNCPoint2[25526] = {X 527.5530, Y 69.8787, Z -3.8333, A 0.000, B 0.000, C 0.000 }
gfCNCPoint2[25527] = {X 525.2751, Y 70.4634, Z -3.8333, A 0.000, B 0.000, C 0.000 }
gfCNCPoint2[25528] = {X 522.9511, Y 70.8245, Z -3.8333, A 0.000, B 0.000, C 0.000 }
gfCNCPoint2[25529] = {X 520.6032, Y 70.9588, Z -3.8333, A 0.000, B 0.000, C 0.000 }
gfCNCPoint2[25530] = {X 519.7998, Y 70.9591, Z -3.8333, A 0.000, B 0.000, C 0.000 }
gfCNCPoint2[25531] = {X 517.4110, Y 70.8403, Z -3.8333, A 0.000, B 0.000, C 0.000 }
gfCNCPoint2[25532] = {X 515.0459, Y 70.4852, Z -3.8333, A 0.000, B 0.000, C 0.000 }
gfCNCPoint2[25533] = {X 512.7276, Y 69.8972, Z -3.8333, A 0.000, B 0.000, C 0.000 }
gfCNCPoint2[25534] = {X 510.4791, Y 69.0821, Z -3.8333, A 0.000, B 0.000, C 0.000 }
gfCNCPoint2[25535] = {X 509.6265, Y 68.7046, Z -3.8333, A 0.000, B 0.000, C 0.000 }
gfCNCPoint2[25536] = {X 508.7892, Y 68.2944, Z -3.8333, A 0.000, B 0.000, C 0.000 }
gfCNCPoint2[25537] = {X 507.1702, Y 68.6593, Z -3.8333, A 0.000, B 0.000, C 0.000 }
gfCNCPoint2[25538] = {X 505.5300, Y 68.9118, Z -3.8333, A 0.000, B 0.000, C 0.000 }
gfCNCPoint2[25539] = {X 504.1117, Y 69.0379, Z -3.8333, A 0.000, B 0.000, C 0.000 }
gfCNCPoint2[25540] = {X 502.6885, Y 69.0800, Z -3.8333, A 0.000, B 0.000, C 0.000 }
gfCNCPoint2[25541] = {X 502.0391, Y 69.0800, Z -3.8333, A 0.000, B 0.000, C 0.000 }
gfCNCPoint2[25542] = {X 501.1774, Y 71.1324, Z -3.8333, A 0.000, B 0.000, C 0.000 }
gfCNCPoint2[25543] = {X 500.1601, Y 73.1123, Z -3.8333, A 0.000, B 0.000, C 0.000 }
gfCNCPoint2[25544] = {X 500.1601, Y 73.6950, Z -3.8333, A 0.000, B 0.000, C 0.000 }
gfCNCPoint2[25545] = {X 507.6816, Y 73.6950, Z -3.8333, A 0.000, B 0.000, C 0.000 }
gfCNCPoint2[25546] = {X 507.6816, Y 76.0950, Z -3.8333, A 0.000, B 0.000, C 0.000 }
gfCNCPoint2[25547] = {X 576.0965, Y 76.0950, Z -3.8333, A 0.000, B 0.000, C 0.000 }
gfCNCPoint2[25548] = {X 576.0965, Y 72.8901, Z -3.8333, A 0.000, B 0.000, C 0.000 }
gfCNCPoint2[25549] = {X 575.7178, Y 72.8147, Z -3.8333, A 0.000, B 0.000, C 0.000 }
gfCNCPoint2[25550] = {X 575.3401, Y 72.7341, Z -3.8333, A 0.000, B 0.000, C 0.000 }
gfCNCPoint2[25551] = {X 573.3201, Y 73.1034, Z -3.8333, A 0.000, B 0.000, C 0.000 }
gfCNCPoint2[25552] = {X 571.2786, Y 73.3258, Z -3.8333, A 0.000, B 0.000, C 0.000 }
gfCNCPoint2[25553] = {X 569.2264, Y 73.4000, Z -3.8333, A 0.000, B 0.000, C 0.000 }
gfCNCPoint2[25554] = {X 562.4443, Y 73.4000, Z -3.8333, A 0.000, B 0.000, C 0.000 }
gfCNCPoint2[25555] = {X 560.3341, Y 73.3215, Z -3.8333, A 0.000, B 0.000, C 0.000 }
gfCNCPoint2[25556] = {X 558.2356, Y 73.0864, Z -3.8333, A 0.000, B 0.000, C 0.000 }
gfCNCPoint2[25557] = {X 556.1604, Y 72.6961, Z -3.8333, A 0.000, B 0.000, C 0.000 }
gfCNCPoint2[25558] = {X 554.1199, Y 72.1526, Z -3.8333, A 0.000, B 0.000, C 0.000 }
gfCNCPoint2[25559] = {X 552.1254, Y 71.4590, Z -3.8333, A 0.000, B 0.000, C 0.000 }
gfCNCPoint2[25560] = {X 549.9760, Y 70.5167, Z -3.8333, A 0.000, B 0.000, C 0.000 }
gfCNCPoint2[25561] = {X 547.9119, Y 69.4002, Z -3.8333, A 0.000, B 0.000, C 0.000 }
gfCNCPoint2[25562] = {X 545.9469, Y 68.1170, Z -3.8333, A 0.000, B 0.000, C 0.000 }
gfCNCPoint2[25563] = {X 544.0946, Y 66.6760, Z -3.8333, A 0.000, B 0.000, C 0.000 }
gfCNCPoint2[25564] = {X 543.8499, Y 66.6772, Z -3.8333, A 0.000, B 0.000, C 0.000 }
gfCNCPoint2[25565] = {X 543.6051, Y 66.6756, Z -3.8333, A 0.000, B 0.000, C 0.000 }
gfCNCPoint2[25566] = {X 529.2679, Y 66.6759, Z -3.8333, A 0.000, B 0.000, C 0.000 }
gfCNCPoint2[25567] = {X 527.1805, Y 67.4788, Z -3.8333, A 0.000, B 0.000, C 0.000 }
gfCNCPoint2[25568] = {X 525.0219, Y 68.0639, Z -3.8333, A 0.000, B 0.000, C 0.000 }
gfCNCPoint2[25569] = {X 522.8149, Y 68.4252, Z -3.8333, A 0.000, B 0.000, C 0.000 }
gfCNCPoint2[25570] = {X 520.5824, Y 68.5589, Z -3.8333, A 0.000, B 0.000, C 0.000 }
gfCNCPoint2[25571] = {X 519.7998, Y 68.5591, Z -3.8333, A 0.000, B 0.000, C 0.000 }
gfCNCPoint2[25572] = {X 517.5593, Y 68.4430, Z -3.8333, A 0.000, B 0.000, C 0.000 }
gfCNCPoint2[25573] = {X 515.3429, Y 68.0961, Z -3.8333, A 0.000, B 0.000, C 0.000 }
gfCNCPoint2[25574] = {X 513.1742, Y 67.5219, Z -3.8333, A 0.000, B 0.000, C 0.000 }
gfCNCPoint2[25575] = {X 511.0764, Y 66.7267, Z -3.8333, A 0.000, B 0.000, C 0.000 }
gfCNCPoint2[25576] = {X 509.0720, Y 65.7189, Z -3.8333, A 0.000, B 0.000, C 0.000 }
gfCNCPoint2[25577] = {X 506.9797, Y 66.2511, Z -3.8333, A 0.000, B 0.000, C 0.000 }
gfCNCPoint2[25578] = {X 504.8448, Y 66.5725, Z -3.8333, A 0.000, B 0.000, C 0.000 }
gfCNCPoint2[25579] = {X 502.6885, Y 66.6800, Z -3.8333, A 0.000, B 0.000, C 0.000 }
gfCNCPoint2[25580] = {X 500.3217, Y 66.6800, Z -3.8333, A 0.000, B 0.000, C 0.000 }
gfCNCPoint2[25581] = {X 499.6230, Y 68.6756, Z -3.8333, A 0.000, B 0.000, C 0.000 }
gfCNCPoint2[25582] = {X 498.7673, Y 70.6090, Z -3.8333, A 0.000, B 0.000, C 0.000 }
gfCNCPoint2[25583] = {X 497.7601, Y 72.4680, Z -3.8333, A 0.000, B 0.000, C 0.000 }
gfCNCPoint2[25584] = {X 497.7602, Y 76.0950, Z -3.8333, A 0.000, B 0.000, C 0.000 }
gfCNCPoint2[25585] = {X 507.6816, Y 76.0950, Z -3.8333, A 0.000, B 0.000, C 0.000 }
gfCNCPoint2[25586] = {X 507.6816, Y 78.4950, Z -3.8333, A 0.000, B 0.000, C 0.000 }
gfCNCPoint2[25587] = {X 578.4965, Y 78.4950, Z -3.8333, A 0.000, B 0.000, C 0.000 }
gfCNCPoint2[25588] = {X 578.4965, Y 70.8313, Z -3.8333, A 0.000, B 0.000, C 0.000 }
gfCNCPoint2[25589] = {X 576.9097, Y 70.5998, Z -3.8333, A 0.000, B 0.000, C 0.000 }
gfCNCPoint2[25590] = {X 575.3401, Y 70.2710, Z -3.8333, A 0.000, B 0.000, C 0.000 }
gfCNCPoint2[25591] = {X 573.3236, Y 70.6751, Z -3.8333, A 0.000, B 0.000, C 0.000 }
gfCNCPoint2[25592] = {X 571.2815, Y 70.9187, Z -3.8333, A 0.000, B 0.000, C 0.000 }
gfCNCPoint2[25593] = {X 569.2264, Y 71.0000, Z -3.8333, A 0.000, B 0.000, C 0.000 }
gfCNCPoint2[25594] = {X 562.4443, Y 71.0000, Z -3.8333, A 0.000, B 0.000, C 0.000 }
gfCNCPoint2[25595] = {X 560.0512, Y 70.8896, Z -3.8333, A 0.000, B 0.000, C 0.000 }
gfCNCPoint2[25596] = {X 557.6784, Y 70.5595, Z -3.8333, A 0.000, B 0.000, C 0.000 }
gfCNCPoint2[25597] = {X 555.3461, Y 70.0123, Z -3.8333, A 0.000, B 0.000, C 0.000 }
gfCNCPoint2[25598] = {X 553.0740, Y 69.2528, Z -3.8333, A 0.000, B 0.000, C 0.000 }
gfCNCPoint2[25599] = {X 550.8815, Y 68.2874, Z -3.8333, A 0.000, B 0.000, C 0.000 }
gfCNCPoint2[25600] = {X 548.7872, Y 67.1243, Z -3.8333, A 0.000, B 0.000, C 0.000 }
gfCNCPoint2[25601] = {X 546.8088, Y 65.7733, Z -3.8333, A 0.000, B 0.000, C 0.000 }
gfCNCPoint2[25602] = {X 544.9631, Y 64.2460, Z -3.8333, A 0.000, B 0.000, C 0.000 }
gfCNCPoint2[25603] = {X 544.2918, Y 64.2725, Z -3.8333, A 0.000, B 0.000, C 0.000 }
gfCNCPoint2[25604] = {X 543.6200, Y 64.2756, Z -3.8333, A 0.000, B 0.000, C 0.000 }
gfCNCPoint2[25605] = {X 528.7428, Y 64.2760, Z -3.8333, A 0.000, B 0.000, C 0.000 }
gfCNCPoint2[25606] = {X 526.7890, Y 65.0780, Z -3.8333, A 0.000, B 0.000, C 0.000 }
gfCNCPoint2[25607] = {X 524.7597, Y 65.6633, Z -3.8333, A 0.000, B 0.000, C 0.000 }
gfCNCPoint2[25608] = {X 522.6789, Y 66.0251, Z -3.8333, A 0.000, B 0.000, C 0.000 }
gfCNCPoint2[25609] = {X 520.5712, Y 66.1589, Z -3.8333, A 0.000, B 0.000, C 0.000 }
gfCNCPoint2[25610] = {X 519.7998, Y 66.1591, Z -3.8333, A 0.000, B 0.000, C 0.000 }
gfCNCPoint2[25611] = {X 517.9641, Y 66.0715, Z -3.8333, A 0.000, B 0.000, C 0.000 }
gfCNCPoint2[25612] = {X 516.1450, Y 65.8096, Z -3.8333, A 0.000, B 0.000, C 0.000 }
gfCNCPoint2[25613] = {X 514.3592, Y 65.3756, Z -3.8333, A 0.000, B 0.000, C 0.000 }
gfCNCPoint2[25614] = {X 512.6228, Y 64.7735, Z -3.8333, A 0.000, B 0.000, C 0.000 }
gfCNCPoint2[25615] = {X 510.9516, Y 64.0089, Z -3.8333, A 0.000, B 0.000, C 0.000 }
gfCNCPoint2[25616] = {X 509.3609, Y 63.0886, Z -3.8333, A 0.000, B 0.000, C 0.000 }
gfCNCPoint2[25617] = {X 507.7389, Y 63.6068, Z -3.8333, A 0.000, B 0.000, C 0.000 }
gfCNCPoint2[25618] = {X 506.0774, Y 63.9798, Z -3.8333, A 0.000, B 0.000, C 0.000 }
gfCNCPoint2[25619] = {X 504.3896, Y 64.2048, Z -3.8333, A 0.000, B 0.000, C 0.000 }
gfCNCPoint2[25620] = {X 502.6885, Y 64.2800, Z -3.8333, A 0.000, B 0.000, C 0.000 }
gfCNCPoint2[25621] = {X 498.4791, Y 64.2800, Z -3.8333, A 0.000, B 0.000, C 0.000 }
gfCNCPoint2[25622] = {X 497.9416, Y 66.2505, Z -3.8333, A 0.000, B 0.000, C 0.000 }
gfCNCPoint2[25623] = {X 497.2390, Y 68.1684, Z -3.8333, A 0.000, B 0.000, C 0.000 }
gfCNCPoint2[25624] = {X 496.3765, Y 70.0198, Z -3.8333, A 0.000, B 0.000, C 0.000 }
gfCNCPoint2[25625] = {X 495.3601, Y 71.7915, Z -3.8333, A 0.000, B 0.000, C 0.000 }
gfCNCPoint2[25626] = {X 495.3602, Y 78.4950, Z -3.8333, A 0.000, B 0.000, C 0.000 }
gfCNCPoint2[25627] = {X 507.6816, Y 78.4950, Z -3.8333, A 0.000, B 0.000, C 0.000 }
gfCNCPoint2[25628] = {X 507.6816, Y 80.8950, Z -3.8333, A 0.000, B 0.000, C 0.000 }
gfCNCPoint2[25629] = {X 580.8965, Y 80.8950, Z -3.8333, A 0.000, B 0.000, C 0.000 }
gfCNCPoint2[25630] = {X 580.8965, Y 68.5934, Z -3.8333, A 0.000, B 0.000, C 0.000 }
gfCNCPoint2[25631] = {X 579.0252, Y 68.4747, Z -3.8333, A 0.000, B 0.000, C 0.000 }
gfCNCPoint2[25632] = {X 577.1691, Y 68.2078, Z -3.8333, A 0.000, B 0.000, C 0.000 }
gfCNCPoint2[25633] = {X 575.3401, Y 67.7943, Z -3.8333, A 0.000, B 0.000, C 0.000 }
gfCNCPoint2[25634] = {X 573.3283, Y 68.2408, Z -3.8333, A 0.000, B 0.000, C 0.000 }
gfCNCPoint2[25635] = {X 571.2852, Y 68.5100, Z -3.8333, A 0.000, B 0.000, C 0.000 }
gfCNCPoint2[25636] = {X 569.2264, Y 68.6000, Z -3.8333, A 0.000, B 0.000, C 0.000 }
gfCNCPoint2[25637] = {X 562.4443, Y 68.6000, Z -3.8333, A 0.000, B 0.000, C 0.000 }
gfCNCPoint2[25638] = {X 560.1443, Y 68.4877, Z -3.8333, A 0.000, B 0.000, C 0.000 }
gfCNCPoint2[25639] = {X 557.8662, Y 68.1517, Z -3.8333, A 0.000, B 0.000, C 0.000 }
gfCNCPoint2[25640] = {X 555.6316, Y 67.5953, Z -3.8333, A 0.000, B 0.000, C 0.000 }
gfCNCPoint2[25641] = {X 553.4619, Y 66.8238, Z -3.8333, A 0.000, B 0.000, C 0.000 }
gfCNCPoint2[25642] = {X 551.3778, Y 65.8445, Z -3.8333, A 0.000, B 0.000, C 0.000 }
gfCNCPoint2[25643] = {X 549.3990, Y 64.6667, Z -3.8333, A 0.000, B 0.000, C 0.000 }
gfCNCPoint2[25644] = {X 547.5444, Y 63.3017, Z -3.8333, A 0.000, B 0.000, C 0.000 }
gfCNCPoint2[25645] = {X 545.8317, Y 61.7625, Z -3.8333, A 0.000, B 0.000, C 0.000 }
gfCNCPoint2[25646] = {X 544.7356, Y 61.8548, Z -3.8333, A 0.000, B 0.000, C 0.000 }
gfCNCPoint2[25647] = {X 543.6359, Y 61.8756, Z -3.8333, A 0.000, B 0.000, C 0.000 }
gfCNCPoint2[25648] = {X 528.1824, Y 61.8760, Z -3.8333, A 0.000, B 0.000, C 0.000 }
gfCNCPoint2[25649] = {X 526.3719, Y 62.6770, Z -3.8333, A 0.000, B 0.000, C 0.000 }
gfCNCPoint2[25650] = {X 524.4808, Y 63.2626, Z -3.8333, A 0.000, B 0.000, C 0.000 }
gfCNCPoint2[25651] = {X 522.5345, Y 63.6248, Z -3.8333, A 0.000, B 0.000, C 0.000 }
gfCNCPoint2[25652] = {X 520.5593, Y 63.7589, Z -3.8333, A 0.000, B 0.000, C 0.000 }
gfCNCPoint2[25653] = {X 519.7998, Y 63.7591, Z -3.8333, A 0.000, B 0.000, C 0.000 }
gfCNCPoint2[25654] = {X 517.9902, Y 63.6618, Z -3.8333, A 0.000, B 0.000, C 0.000 }
gfCNCPoint2[25655] = {X 516.2015, Y 63.3711, Z -3.8333, A 0.000, B 0.000, C 0.000 }
gfCNCPoint2[25656] = {X 514.4543, Y 62.8904, Z -3.8333, A 0.000, B 0.000, C 0.000 }
gfCNCPoint2[25657] = {X 512.7687, Y 62.2251, Z -3.8333, A 0.000, B 0.000, C 0.000 }
gfCNCPoint2[25658] = {X 511.1641, Y 61.3829, Z -3.8333, A 0.000, B 0.000, C 0.000 }
gfCNCPoint2[25659] = {X 509.6590, Y 60.3735, Z -3.8333, A 0.000, B 0.000, C 0.000 }
gfCNCPoint2[25660] = {X 507.9866, Y 61.0270, Z -3.8333, A 0.000, B 0.000, C 0.000 }
gfCNCPoint2[25661] = {X 506.2542, Y 61.4991, Z -3.8333, A 0.000, B 0.000, C 0.000 }
gfCNCPoint2[25662] = {X 504.4815, Y 61.7845, Z -3.8333, A 0.000, B 0.000, C 0.000 }
gfCNCPoint2[25663] = {X 502.6885, Y 61.8800, Z -3.8333, A 0.000, B 0.000, C 0.000 }
gfCNCPoint2[25664] = {X 496.4789, Y 61.8800, Z -3.8333, A 0.000, B 0.000, C 0.000 }
gfCNCPoint2[25665] = {X 496.1192, Y 63.8333, Z -3.8333, A 0.000, B 0.000, C 0.000 }
gfCNCPoint2[25666] = {X 495.5822, Y 65.7454, Z -3.8333, A 0.000, B 0.000, C 0.000 }
gfCNCPoint2[25667] = {X 494.8725, Y 67.6004, Z -3.8333, A 0.000, B 0.000, C 0.000 }
gfCNCPoint2[25668] = {X 493.9960, Y 69.3827, Z -3.8333, A 0.000, B 0.000, C 0.000 }
gfCNCPoint2[25669] = {X 492.9601, Y 71.0773, Z -3.8333, A 0.000, B 0.000, C 0.000 }
gfCNCPoint2[25670] = {X 492.9602, Y 80.8950, Z -3.8333, A 0.000, B 0.000, C 0.000 }
gfCNCPoint2[25671] = {X 507.6816, Y 80.8950, Z -3.8333, A 0.000, B 0.000, C 0.000 }
gfCNCPoint2[25672] = {X 507.6816, Y 83.2950, Z -3.8333, A 0.000, B 0.000, C 0.000 }
gfCNCPoint2[25673] = {X 583.2965, Y 83.2950, Z -3.8333, A 0.000, B 0.000, C 0.000 }
gfCNCPoint2[25674] = {X 583.2965, Y 66.1198, Z -3.8333, A 0.000, B 0.000, C 0.000 }
gfCNCPoint2[25675] = {X 581.2872, Y 66.1993, Z -3.8333, A 0.000, B 0.000, C 0.000 }
gfCNCPoint2[25676] = {X 579.2793, Y 66.0882, Z -3.8333, A 0.000, B 0.000, C 0.000 }
gfCNCPoint2[25677] = {X 577.2910, Y 65.7873, Z -3.8333, A 0.000, B 0.000, C 0.000 }
gfCNCPoint2[25678] = {X 575.3401, Y 65.2993, Z -3.8333, A 0.000, B 0.000, C 0.000 }
gfCNCPoint2[25679] = {X 573.3348, Y 65.7981, Z -3.8333, A 0.000, B 0.000, C 0.000 }
gfCNCPoint2[25680] = {X 571.2904, Y 66.0993, Z -3.8333, A 0.000, B 0.000, C 0.000 }
gfCNCPoint2[25681] = {X 569.2264, Y 66.2000, Z -3.8333, A 0.000, B 0.000, C 0.000 }
gfCNCPoint2[25682] = {X 562.4443, Y 66.2000, Z -3.8333, A 0.000, B 0.000, C 0.000 }
gfCNCPoint2[25683] = {X 560.2303, Y 66.0841, Z -3.8333, A 0.000, B 0.000, C 0.000 }
gfCNCPoint2[25684] = {X 558.0405, Y 65.7376, Z -3.8333, A 0.000, B 0.000, C 0.000 }
gfCNCPoint2[25685] = {X 555.8988, Y 65.1642, Z -3.8333, A 0.000, B 0.000, C 0.000 }
gfCNCPoint2[25686] = {X 553.8287, Y 64.3704, Z -3.8333, A 0.000, B 0.000, C 0.000 }
gfCNCPoint2[25687] = {X 551.8529, Y 63.3647, Z -3.8333, A 0.000, B 0.000, C 0.000 }
gfCNCPoint2[25688] = {X 549.9929, Y 62.1582, Z -3.8333, A 0.000, B 0.000, C 0.000 }
gfCNCPoint2[25689] = {X 548.2691, Y 60.7640, Z -3.8333, A 0.000, B 0.000, C 0.000 }
gfCNCPoint2[25690] = {X 546.7003, Y 59.1974, Z -3.8333, A 0.000, B 0.000, C 0.000 }
gfCNCPoint2[25691] = {X 545.1840, Y 59.4172, Z -3.8333, A 0.000, B 0.000, C 0.000 }
gfCNCPoint2[25692] = {X 543.6529, Y 59.4756, Z -3.8333, A 0.000, B 0.000, C 0.000 }
gfCNCPoint2[25693] = {X 527.5783, Y 59.4760, Z -3.8333, A 0.000, B 0.000, C 0.000 }
gfCNCPoint2[25694] = {X 525.9210, Y 60.2766, Z -3.8333, A 0.000, B 0.000, C 0.000 }
gfCNCPoint2[25695] = {X 524.1763, Y 60.8629, Z -3.8333, A 0.000, B 0.000, C 0.000 }
gfCNCPoint2[25696] = {X 522.3718, Y 61.2256, Z -3.8333, A 0.000, B 0.000, C 0.000 }
gfCNCPoint2[25697] = {X 520.5361, Y 61.3590, Z -3.8333, A 0.000, B 0.000, C 0.000 }
gfCNCPoint2[25698] = {X 519.7998, Y 61.3591, Z -3.8333, A 0.000, B 0.000, C 0.000 }
gfCNCPoint2[25699] = {X 518.0043, Y 61.2474, Z -3.8333, A 0.000, B 0.000, C 0.000 }
gfCNCPoint2[25700] = {X 516.2365, Y 60.9138, Z -3.8333, A 0.000, B 0.000, C 0.000 }
gfCNCPoint2[25701] = {X 514.5237, Y 60.3637, Z -3.8333, A 0.000, B 0.000, C 0.000 }
gfCNCPoint2[25702] = {X 512.8923, Y 59.6054, Z -3.8333, A 0.000, B 0.000, C 0.000 }
gfCNCPoint2[25703] = {X 511.3676, Y 58.6507, Z -3.8333, A 0.000, B 0.000, C 0.000 }
gfCNCPoint2[25704] = {X 509.9730, Y 57.5142, Z -3.8333, A 0.000, B 0.000, C 0.000 }
gfCNCPoint2[25705] = {X 508.6156, Y 58.2113, Z -3.8333, A 0.000, B 0.000, C 0.000 }
gfCNCPoint2[25706] = {X 507.1924, Y 58.7617, Z -3.8333, A 0.000, B 0.000, C 0.000 }
gfCNCPoint2[25707] = {X 505.7192, Y 59.1593, Z -3.8333, A 0.000, B 0.000, C 0.000 }
gfCNCPoint2[25708] = {X 504.2123, Y 59.3996, Z -3.8333, A 0.000, B 0.000, C 0.000 }
gfCNCPoint2[25709] = {X 502.6885, Y 59.4800, Z -3.8333, A 0.000, B 0.000, C 0.000 }
gfCNCPoint2[25710] = {X 496.2450, Y 59.4800, Z -3.8333, A 0.000, B 0.000, C 0.000 }
gfCNCPoint2[25711] = {X 495.2580, Y 59.4463, Z -3.8333, A 0.000, B 0.000, C 0.000 }
gfCNCPoint2[25712] = {X 494.2756, Y 59.3454, Z -3.8333, A 0.000, B 0.000, C 0.000 }
gfCNCPoint2[25713] = {X 494.1342, Y 61.3006, Z -3.8333, A 0.000, B 0.000, C 0.000 }
gfCNCPoint2[25714] = {X 493.7950, Y 63.2313, Z -3.8333, A 0.000, B 0.000, C 0.000 }
gfCNCPoint2[25715] = {X 493.2615, Y 65.1176, Z -3.8333, A 0.000, B 0.000, C 0.000 }
gfCNCPoint2[25716] = {X 492.5392, Y 66.9399, Z -3.8333, A 0.000, B 0.000, C 0.000 }
gfCNCPoint2[25717] = {X 491.6356, Y 68.6795, Z -3.8333, A 0.000, B 0.000, C 0.000 }
gfCNCPoint2[25718] = {X 490.5601, Y 70.3184, Z -3.8333, A 0.000, B 0.000, C 0.000 }
gfCNCPoint2[25719] = {X 490.5603, Y 83.2950, Z -3.8333, A 0.000, B 0.000, C 0.000 }
gfCNCPoint2[25720] = {X 507.6816, Y 83.2950, Z -3.8333, A 0.000, B 0.000, C 0.000 }
gfCNCPoint2[25721] = {X 507.6816, Y 85.6950, Z -3.8333, A 0.000, B 0.000, C 0.000 }
gfCNCPoint2[25722] = {X 585.6965, Y 85.6950, Z -3.8333, A 0.000, B 0.000, C 0.000 }
gfCNCPoint2[25723] = {X 585.6965, Y 63.3150, Z -3.8333, A 0.000, B 0.000, C 0.000 }
gfCNCPoint2[25724] = {X 584.3995, Y 63.5678, Z -3.8333, A 0.000, B 0.000, C 0.000 }
gfCNCPoint2[25725] = {X 583.0879, Y 63.7288, Z -3.8333, A 0.000, B 0.000, C 0.000 }
gfCNCPoint2[25726] = {X 581.1242, Y 63.7971, Z -3.8333, A 0.000, B 0.000, C 0.000 }
gfCNCPoint2[25727] = {X 579.1642, Y 63.6600, Z -3.8333, A 0.000, B 0.000, C 0.000 }
gfCNCPoint2[25728] = {X 577.2291, Y 63.3191, Z -3.8333, A 0.000, B 0.000, C 0.000 }
gfCNCPoint2[25729] = {X 575.3401, Y 62.7781, Z -3.8333, A 0.000, B 0.000, C 0.000 }
gfCNCPoint2[25730] = {X 573.3441, Y 63.3435, Z -3.8333, A 0.000, B 0.000, C 0.000 }
gfCNCPoint2[25731] = {X 571.2979, Y 63.6855, Z -3.8333, A 0.000, B 0.000, C 0.000 }
gfCNCPoint2[25732] = {X 569.2264, Y 63.8000, Z -3.8333, A 0.000, B 0.000, C 0.000 }
gfCNCPoint2[25733] = {X 562.4443, Y 63.8000, Z -3.8333, A 0.000, B 0.000, C 0.000 }
gfCNCPoint2[25734] = {X 560.5407, Y 63.7034, Z -3.8333, A 0.000, B 0.000, C 0.000 }
gfCNCPoint2[25735] = {X 558.6567, Y 63.4145, Z -3.8333, A 0.000, B 0.000, C 0.000 }
gfCNCPoint2[25736] = {X 556.8117, Y 62.9364, Z -3.8333, A 0.000, B 0.000, C 0.000 }
gfCNCPoint2[25737] = {X 555.0245, Y 62.2739, Z -3.8333, A 0.000, B 0.000, C 0.000 }
gfCNCPoint2[25738] = {X 553.3136, Y 61.4338, Z -3.8333, A 0.000, B 0.000, C 0.000 }
gfCNCPoint2[25739] = {X 551.6966, Y 60.4249, Z -3.8333, A 0.000, B 0.000, C 0.000 }
gfCNCPoint2[25740] = {X 550.1900, Y 59.2573, Z -3.8333, A 0.000, B 0.000, C 0.000 }
gfCNCPoint2[25741] = {X 548.8094, Y 57.9433, Z -3.8333, A 0.000, B 0.000, C 0.000 }
gfCNCPoint2[25742] = {X 547.5689, Y 56.4962, Z -3.8333, A 0.000, B 0.000, C 0.000 }
gfCNCPoint2[25743] = {X 546.2935, Y 56.8311, Z -3.8333, A 0.000, B 0.000, C 0.000 }
gfCNCPoint2[25744] = {X 544.9891, Y 57.0250, Z -3.8333, A 0.000, B 0.000, C 0.000 }
gfCNCPoint2[25745] = {X 543.6714, Y 57.0756, Z -3.8333, A 0.000, B 0.000, C 0.000 }
gfCNCPoint2[25746] = {X 526.9187, Y 57.0760, Z -3.8333, A 0.000, B 0.000, C 0.000 }
gfCNCPoint2[25747] = {X 525.4306, Y 57.8757, Z -3.8333, A 0.000, B 0.000, C 0.000 }
gfCNCPoint2[25748] = {X 523.8467, Y 58.4629, Z -3.8333, A 0.000, B 0.000, C 0.000 }
gfCNCPoint2[25749] = {X 522.1969, Y 58.8263, Z -3.8333, A 0.000, B 0.000, C 0.000 }
gfCNCPoint2[25750] = {X 520.5128, Y 58.9591, Z -3.8333, A 0.000, B 0.000, C 0.000 }
gfCNCPoint2[25751] = {X 519.7998, Y 58.9591, Z -3.8333, A 0.000, B 0.000, C 0.000 }
gfCNCPoint2[25752] = {X 518.2467, Y 58.8589, Z -3.8333, A 0.000, B 0.000, C 0.000 }
gfCNCPoint2[25753] = {X 516.7195, Y 58.5598, Z -3.8333, A 0.000, B 0.000, C 0.000 }
gfCNCPoint2[25754] = {X 515.2433, Y 58.0668, Z -3.8333, A 0.000, B 0.000, C 0.000 }
gfCNCPoint2[25755] = {X 513.8428, Y 57.3882, Z -3.8333, A 0.000, B 0.000, C 0.000 }
gfCNCPoint2[25756] = {X 512.5411, Y 56.5351, Z -3.8333, A 0.000, B 0.000, C 0.000 }
gfCNCPoint2[25757] = {X 511.3600, Y 55.5218, Z -3.8333, A 0.000, B 0.000, C 0.000 }
gfCNCPoint2[25758] = {X 510.3189, Y 54.3650, Z -3.8333, A 0.000, B 0.000, C 0.000 }
gfCNCPoint2[25759] = {X 508.9711, Y 55.3177, Z -3.8333, A 0.000, B 0.000, C 0.000 }
gfCNCPoint2[25760] = {X 507.5060, Y 56.0778, Z -3.8333, A 0.000, B 0.000, C 0.000 }
gfCNCPoint2[25761] = {X 505.9510, Y 56.6311, Z -3.8333, A 0.000, B 0.000, C 0.000 }
gfCNCPoint2[25762] = {X 504.3351, Y 56.9672, Z -3.8333, A 0.000, B 0.000, C 0.000 }
gfCNCPoint2[25763] = {X 502.6885, Y 57.0800, Z -3.8333, A 0.000, B 0.000, C 0.000 }
gfCNCPoint2[25764] = {X 496.2450, Y 57.0800, Z -3.8333, A 0.000, B 0.000, C 0.000 }
gfCNCPoint2[25765] = {X 495.4216, Y 57.0519, Z -3.8333, A 0.000, B 0.000, C 0.000 }
gfCNCPoint2[25766] = {X 494.6020, Y 56.9677, Z -3.8333, A 0.000, B 0.000, C 0.000 }
gfCNCPoint2[25767] = {X 493.1719, Y 56.6826, Z -3.8333, A 0.000, B 0.000, C 0.000 }
gfCNCPoint2[25768] = {X 491.7866, Y 56.2272, Z -3.8333, A 0.000, B 0.000, C 0.000 }
gfCNCPoint2[25769] = {X 491.8566, Y 57.1124, Z -3.8333, A 0.000, B 0.000, C 0.000 }
gfCNCPoint2[25770] = {X 491.8800, Y 58.0000, Z -3.8333, A 0.000, B 0.000, C 0.000 }
gfCNCPoint2[25771] = {X 491.8794, Y 59.0735, Z -3.8333, A 0.000, B 0.000, C 0.000 }
gfCNCPoint2[25772] = {X 491.8781, Y 59.1839, Z -3.8333, A 0.000, B 0.000, C 0.000 }
gfCNCPoint2[25773] = {X 491.8762, Y 59.2942, Z -3.8333, A 0.000, B 0.000, C 0.000 }
gfCNCPoint2[25774] = {X 491.7363, Y 61.1318, Z -3.8333, A 0.000, B 0.000, C 0.000 }
gfCNCPoint2[25775] = {X 491.3970, Y 62.9432, Z -3.8333, A 0.000, B 0.000, C 0.000 }
gfCNCPoint2[25776] = {X 490.8622, Y 64.7069, Z -3.8333, A 0.000, B 0.000, C 0.000 }
gfCNCPoint2[25777] = {X 490.1383, Y 66.4017, Z -3.8333, A 0.000, B 0.000, C 0.000 }
gfCNCPoint2[25778] = {X 489.2340, Y 68.0075, Z -3.8333, A 0.000, B 0.000, C 0.000 }
gfCNCPoint2[25779] = {X 488.1601, Y 69.5051, Z -3.8333, A 0.000, B 0.000, C 0.000 }
gfCNCPoint2[25780] = {X 488.1603, Y 85.6950, Z -3.8333, A 0.000, B 0.000, C 0.000 }
gfCNCPoint2[25781] = {X 507.6816, Y 85.6950, Z -3.8333, A 0.000, B 0.000, C 0.000 }
gfCNCPoint2[25782] = {X 507.6816, Y 88.0950, Z -3.8333, A 0.000, B 0.000, C 0.000 }
gfCNCPoint2[25783] = {X 588.0965, Y 88.0950, Z -3.8333, A 0.000, B 0.000, C 0.000 }
gfCNCPoint2[25784] = {X 588.0965, Y 60.4644, Z -3.8333, A 0.000, B 0.000, C 0.000 }
gfCNCPoint2[25785] = {X 587.7998, Y 60.3564, Z -3.8333, A 0.000, B 0.000, C 0.000 }
gfCNCPoint2[25786] = {X 587.5052, Y 60.2427, Z -3.8333, A 0.000, B 0.000, C 0.000 }
gfCNCPoint2[25787] = {X 586.3439, Y 60.6540, Z -3.8333, A 0.000, B 0.000, C 0.000 }
gfCNCPoint2[25788] = {X 585.1549, Y 60.9769, Z -3.8333, A 0.000, B 0.000, C 0.000 }
gfCNCPoint2[25789] = {X 583.5153, Y 61.2699, Z -3.8333, A 0.000, B 0.000, C 0.000 }
gfCNCPoint2[25790] = {X 581.8543, Y 61.3951, Z -3.8333, A 0.000, B 0.000, C 0.000 }
gfCNCPoint2[25791] = {X 580.1892, Y 61.3512, Z -3.8333, A 0.000, B 0.000, C 0.000 }
gfCNCPoint2[25792] = {X 578.5372, Y 61.1386, Z -3.8333, A 0.000, B 0.000, C 0.000 }
gfCNCPoint2[25793] = {X 576.9153, Y 60.7595, Z -3.8333, A 0.000, B 0.000, C 0.000 }
gfCNCPoint2[25794] = {X 575.3401, Y 60.2178, Z -3.8333, A 0.000, B 0.000, C 0.000 }
gfCNCPoint2[25795] = {X 573.8611, Y 60.7315, Z -3.8333, A 0.000, B 0.000, C 0.000 }
gfCNCPoint2[25796] = {X 572.3399, Y 61.1017, Z -3.8333, A 0.000, B 0.000, C 0.000 }
gfCNCPoint2[25797] = {X 570.7903, Y 61.3253, Z -3.8333, A 0.000, B 0.000, C 0.000 }
gfCNCPoint2[25798] = {X 569.2264, Y 61.4000, Z -3.8333, A 0.000, B 0.000, C 0.000 }
gfCNCPoint2[25799] = {X 562.4443, Y 61.4000, Z -3.8333, A 0.000, B 0.000, C 0.000 }
gfCNCPoint2[25800] = {X 560.5828, Y 61.2940, Z -3.8333, A 0.000, B 0.000, C 0.000 }
gfCNCPoint2[25801] = {X 558.7454, Y 60.9774, Z -3.8333, A 0.000, B 0.000, C 0.000 }
gfCNCPoint2[25802] = {X 556.9558, Y 60.4543, Z -3.8333, A 0.000, B 0.000, C 0.000 }
gfCNCPoint2[25803] = {X 555.2371, Y 59.7315, Z -3.8333, A 0.000, B 0.000, C 0.000 }
gfCNCPoint2[25804] = {X 553.6116, Y 58.8182, Z -3.8333, A 0.000, B 0.000, C 0.000 }
gfCNCPoint2[25805] = {X 552.1002, Y 57.7264, Z -3.8333, A 0.000, B 0.000, C 0.000 }
gfCNCPoint2[25806] = {X 550.7226, Y 56.4700, Z -3.8333, A 0.000, B 0.000, C 0.000 }
gfCNCPoint2[25807] = {X 549.4964, Y 55.0654, Z -3.8333, A 0.000, B 0.000, C 0.000 }
gfCNCPoint2[25808] = {X 548.4376, Y 53.5307, Z -3.8333, A 0.000, B 0.000, C 0.000 }
gfCNCPoint2[25809] = {X 547.3158, Y 54.0423, Z -3.8333, A 0.000, B 0.000, C 0.000 }
gfCNCPoint2[25810] = {X 546.1381, Y 54.4071, Z -3.8333, A 0.000, B 0.000, C 0.000 }
gfCNCPoint2[25811] = {X 544.9235, Y 54.6194, Z -3.8333, A 0.000, B 0.000, C 0.000 }
gfCNCPoint2[25812] = {X 543.6919, Y 54.6756, Z -3.8333, A 0.000, B 0.000, C 0.000 }
gfCNCPoint2[25813] = {X 526.1843, Y 54.6760, Z -3.8333, A 0.000, B 0.000, C 0.000 }
gfCNCPoint2[25814] = {X 524.8902, Y 55.4727, Z -3.8333, A 0.000, B 0.000, C 0.000 }
gfCNCPoint2[25815] = {X 523.4889, Y 56.0606, Z -3.8333, A 0.000, B 0.000, C 0.000 }
gfCNCPoint2[25816] = {X 522.0138, Y 56.4256, Z -3.8333, A 0.000, B 0.000, C 0.000 }
gfCNCPoint2[25817] = {X 520.5000, Y 56.5591, Z -3.8333, A 0.000, B 0.000, C 0.000 }
gfCNCPoint2[25818] = {X 519.7998, Y 56.5591, Z -3.8333, A 0.000, B 0.000, C 0.000 }
gfCNCPoint2[25819] = {X 518.3493, Y 56.4498, Z -3.8333, A 0.000, B 0.000, C 0.000 }
gfCNCPoint2[25820] = {X 516.9316, Y 56.1244, Z -3.8333, A 0.000, B 0.000, C 0.000 }
gfCNCPoint2[25821] = {X 515.5787, Y 55.5903, Z -3.8333, A 0.000, B 0.000, C 0.000 }
gfCNCPoint2[25822] = {X 514.3210, Y 54.8595, Z -3.8333, A 0.000, B 0.000, C 0.000 }
gfCNCPoint2[25823] = {X 513.1871, Y 53.9484, Z -3.8333, A 0.000, B 0.000, C 0.000 }
gfCNCPoint2[25824] = {X 512.2025, Y 52.8778, Z -3.8333, A 0.000, B 0.000, C 0.000 }
gfCNCPoint2[25825] = {X 511.3855, Y 51.6648, Z -3.8333, A 0.000, B 0.000, C 0.000 }
gfCNCPoint2[25826] = {X 510.7606, Y 50.3426, Z -3.8333, A 0.000, B 0.000, C 0.000 }
gfCNCPoint2[25827] = {X 509.8636, Y 51.4977, Z -3.8333, A 0.000, B 0.000, C 0.000 }
gfCNCPoint2[25828] = {X 508.8029, Y 52.5044, Z -3.8333, A 0.000, B 0.000, C 0.000 }
gfCNCPoint2[25829] = {X 507.7229, Y 53.2678, Z -3.8333, A 0.000, B 0.000, C 0.000 }
gfCNCPoint2[25830] = {X 506.5489, Y 53.8769, Z -3.8333, A 0.000, B 0.000, C 0.000 }
gfCNCPoint2[25831] = {X 505.3028, Y 54.3203, Z -3.8333, A 0.000, B 0.000, C 0.000 }
gfCNCPoint2[25832] = {X 504.0080, Y 54.5896, Z -3.8333, A 0.000, B 0.000, C 0.000 }
gfCNCPoint2[25833] = {X 502.6885, Y 54.6800, Z -3.8333, A 0.000, B 0.000, C 0.000 }
gfCNCPoint2[25834] = {X 496.2450, Y 54.6800, Z -3.8333, A 0.000, B 0.000, C 0.000 }
gfCNCPoint2[25835] = {X 495.0285, Y 54.6033, Z -3.8333, A 0.000, B 0.000, C 0.000 }
gfCNCPoint2[25836] = {X 493.8313, Y 54.3742, Z -3.8333, A 0.000, B 0.000, C 0.000 }
gfCNCPoint2[25837] = {X 492.6724, Y 53.9966, Z -3.8333, A 0.000, B 0.000, C 0.000 }
gfCNCPoint2[25838] = {X 491.4451, Y 53.4062, Z -3.8333, A 0.000, B 0.000, C 0.000 }
gfCNCPoint2[25839] = {X 490.3129, Y 52.6493, Z -3.8333, A 0.000, B 0.000, C 0.000 }
gfCNCPoint2[25840] = {X 489.2980, Y 51.7410, Z -3.8333, A 0.000, B 0.000, C 0.000 }
gfCNCPoint2[25841] = {X 488.8683, Y 52.1573, Z -3.8333, A 0.000, B 0.000, C 0.000 }
gfCNCPoint2[25842] = {X 488.4137, Y 52.5463, Z -3.8333, A 0.000, B 0.000, C 0.000 }
gfCNCPoint2[25843] = {X 488.8649, Y 53.8245, Z -3.8333, A 0.000, B 0.000, C 0.000 }
gfCNCPoint2[25844] = {X 489.1946, Y 55.1393, Z -3.8333, A 0.000, B 0.000, C 0.000 }
gfCNCPoint2[25845] = {X 489.3999, Y 56.4792, Z -3.8333, A 0.000, B 0.000, C 0.000 }
gfCNCPoint2[25846] = {X 489.4600, Y 57.2386, Z -3.8333, A 0.000, B 0.000, C 0.000 }
gfCNCPoint2[25847] = {X 489.4800, Y 58.0000, Z -3.8333, A 0.000, B 0.000, C 0.000 }
gfCNCPoint2[25848] = {X 489.4795, Y 59.0537, Z -3.8333, A 0.000, B 0.000, C 0.000 }
gfCNCPoint2[25849] = {X 489.3596, Y 60.7978, Z -3.8333, A 0.000, B 0.000, C 0.000 }
gfCNCPoint2[25850] = {X 489.0303, Y 62.5147, Z -3.8333, A 0.000, B 0.000, C 0.000 }
gfCNCPoint2[25851] = {X 488.4965, Y 64.1795, Z -3.8333, A 0.000, B 0.000, C 0.000 }
gfCNCPoint2[25852] = {X 487.7660, Y 65.7678, Z -3.8333, A 0.000, B 0.000, C 0.000 }
gfCNCPoint2[25853] = {X 486.8494, Y 67.2565, Z -3.8333, A 0.000, B 0.000, C 0.000 }
gfCNCPoint2[25854] = {X 485.7601, Y 68.6238, Z -3.8333, A 0.000, B 0.000, C 0.000 }
gfCNCPoint2[25855] = {X 485.7603, Y 87.3796, Z -3.8333, A 0.000, B 0.000, C 0.000 }
gfCNCPoint2[25856] = {X 486.0682, Y 87.7324, Z -3.8333, A 0.000, B 0.000, C 0.000 }
gfCNCPoint2[25857] = {X 486.3646, Y 88.0950, Z -3.8333, A 0.000, B 0.000, C 0.000 }
gfCNCPoint2[25858] = {X 507.6816, Y 88.0950, Z -3.8333, A 0.000, B 0.000, C 0.000 }
gfCNCPoint2[25859] = {X 507.6816, Y 90.4950, Z -3.8333, A 0.000, B 0.000, C 0.000 }
gfCNCPoint2[25860] = {X 590.4965, Y 90.4950, Z -3.8333, A 0.000, B 0.000, C 0.000 }
gfCNCPoint2[25861] = {X 590.4965, Y 58.6615, Z -3.8333, A 0.000, B 0.000, C 0.000 }
gfCNCPoint2[25862] = {X 588.9715, Y 58.2279, Z -3.8333, A 0.000, B 0.000, C 0.000 }
gfCNCPoint2[25863] = {X 587.5052, Y 57.6246, Z -3.8333, A 0.000, B 0.000, C 0.000 }
gfCNCPoint2[25864] = {X 585.8387, Y 58.2956, Z -3.8333, A 0.000, B 0.000, C 0.000 }
gfCNCPoint2[25865] = {X 584.0999, Y 58.7477, Z -3.8333, A 0.000, B 0.000, C 0.000 }
gfCNCPoint2[25866] = {X 582.3176, Y 58.9733, Z -3.8333, A 0.000, B 0.000, C 0.000 }
gfCNCPoint2[25867] = {X 580.5210, Y 58.9689, Z -3.8333, A 0.000, B 0.000, C 0.000 }
gfCNCPoint2[25868] = {X 578.7398, Y 58.7344, Z -3.8333, A 0.000, B 0.000, C 0.000 }
gfCNCPoint2[25869] = {X 577.0034, Y 58.2738, Z -3.8333, A 0.000, B 0.000, C 0.000 }
gfCNCPoint2[25870] = {X 575.3401, Y 57.5945, Z -3.8333, A 0.000, B 0.000, C 0.000 }
gfCNCPoint2[25871] = {X 573.8813, Y 58.2035, Z -3.8333, A 0.000, B 0.000, C 0.000 }
gfCNCPoint2[25872] = {X 572.3630, Y 58.6441, Z -3.8333, A 0.000, B 0.000, C 0.000 }
gfCNCPoint2[25873] = {X 570.8048, Y 58.9107, Z -3.8333, A 0.000, B 0.000, C 0.000 }
gfCNCPoint2[25874] = {X 569.2264, Y 59.0000, Z -3.8333, A 0.000, B 0.000, C 0.000 }
gfCNCPoint2[25875] = {X 562.4443, Y 59.0000, Z -3.8333, A 0.000, B 0.000, C 0.000 }
gfCNCPoint2[25876] = {X 560.6576, Y 58.8855, Z -3.8333, A 0.000, B 0.000, C 0.000 }
gfCNCPoint2[25877] = {X 558.9002, Y 58.5440, Z -3.8333, A 0.000, B 0.000, C 0.000 }
gfCNCPoint2[25878] = {X 557.2007, Y 57.9809, Z -3.8333, A 0.000, B 0.000, C 0.000 }
gfCNCPoint2[25879] = {X 555.5869, Y 57.2056, Z -3.8333, A 0.000, B 0.000, C 0.000 }
gfCNCPoint2[25880] = {X 554.0853, Y 56.2306, Z -3.8333, A 0.000, B 0.000, C 0.000 }
gfCNCPoint2[25881] = {X 552.7204, Y 55.0720, Z -3.8333, A 0.000, B 0.000, C 0.000 }
gfCNCPoint2[25882] = {X 551.5145, Y 53.7487, Z -3.8333, A 0.000, B 0.000, C 0.000 }
gfCNCPoint2[25883] = {X 550.4874, Y 52.2823, Z -3.8333, A 0.000, B 0.000, C 0.000 }
gfCNCPoint2[25884] = {X 549.8376, Y 51.0887, Z -3.8333, A 0.000, B 0.000, C 0.000 }
gfCNCPoint2[25885] = {X 549.3067, Y 49.8376, Z -3.8333, A 0.000, B 0.000, C 0.000 }
gfCNCPoint2[25886] = {X 548.3753, Y 50.7144, Z -3.8333, A 0.000, B 0.000, C 0.000 }
gfCNCPoint2[25887] = {X 547.3049, Y 51.4148, Z -3.8333, A 0.000, B 0.000, C 0.000 }
gfCNCPoint2[25888] = {X 546.1634, Y 51.9057, Z -3.8333, A 0.000, B 0.000, C 0.000 }
gfCNCPoint2[25889] = {X 544.9551, Y 52.1954, Z -3.8333, A 0.000, B 0.000, C 0.000 }
gfCNCPoint2[25890] = {X 543.7151, Y 52.2756, Z -3.8333, A 0.000, B 0.000, C 0.000 }
gfCNCPoint2[25891] = {X 525.3421, Y 52.2760, Z -3.8333, A 0.000, B 0.000, C 0.000 }
gfCNCPoint2[25892] = {X 524.2750, Y 53.0676, Z -3.8333, A 0.000, B 0.000, C 0.000 }
gfCNCPoint2[25893] = {X 523.0840, Y 53.6566, Z -3.8333, A 0.000, B 0.000, C 0.000 }
gfCNCPoint2[25894] = {X 521.8073, Y 54.0244, Z -3.8333, A 0.000, B 0.000, C 0.000 }
gfCNCPoint2[25895] = {X 520.4855, Y 54.1591, Z -3.8333, A 0.000, B 0.000, C 0.000 }
gfCNCPoint2[25896] = {X 519.7998, Y 54.1591, Z -3.8333, A 0.000, B 0.000, C 0.000 }
gfCNCPoint2[25897] = {X 518.5529, Y 54.0515, Z -3.8333, A 0.000, B 0.000, C 0.000 }
gfCNCPoint2[25898] = {X 517.3428, Y 53.7320, Z -3.8333, A 0.000, B 0.000, C 0.000 }
gfCNCPoint2[25899] = {X 516.2054, Y 53.2099, Z -3.8333, A 0.000, B 0.000, C 0.000 }
gfCNCPoint2[25900] = {X 515.1742, Y 52.5007, Z -3.8333, A 0.000, B 0.000, C 0.000 }
gfCNCPoint2[25901] = {X 514.2797, Y 51.6254, Z -3.8333, A 0.000, B 0.000, C 0.000 }
gfCNCPoint2[25902] = {X 513.5483, Y 50.6098, Z -3.8333, A 0.000, B 0.000, C 0.000 }
gfCNCPoint2[25903] = {X 513.0017, Y 49.4839, Z -3.8333, A 0.000, B 0.000, C 0.000 }
gfCNCPoint2[25904] = {X 512.7353, Y 48.6374, Z -3.8333, A 0.000, B 0.000, C 0.000 }
gfCNCPoint2[25905] = {X 512.5739, Y 47.7649, Z -3.8333, A 0.000, B 0.000, C 0.000 }
gfCNCPoint2[25906] = {X 512.5198, Y 46.8791, Z -3.8333, A 0.000, B 0.000, C 0.000 }
gfCNCPoint2[25907] = {X 512.5198, Y 39.9011, Z -3.8333, A 0.000, B 0.000, C 0.000 }
gfCNCPoint2[25908] = {X 512.5807, Y 38.9612, Z -3.8333, A 0.000, B 0.000, C 0.000 }
gfCNCPoint2[25909] = {X 512.7625, Y 38.0370, Z -3.8333, A 0.000, B 0.000, C 0.000 }
gfCNCPoint2[25910] = {X 513.0621, Y 37.1440, Z -3.8333, A 0.000, B 0.000, C 0.000 }
gfCNCPoint2[25911] = {X 513.5576, Y 36.1549, Z -3.8333, A 0.000, B 0.000, C 0.000 }
gfCNCPoint2[25912] = {X 514.1973, Y 35.2524, Z -3.8333, A 0.000, B 0.000, C 0.000 }
gfCNCPoint2[25913] = {X 514.9664, Y 34.4571, Z -3.8333, A 0.000, B 0.000, C 0.000 }
gfCNCPoint2[25914] = {X 515.8471, Y 33.7876, Z -3.8333, A 0.000, B 0.000, C 0.000 }
gfCNCPoint2[25915] = {X 513.2409, Y 29.7568, Z -3.8333, A 0.000, B 0.000, C 0.000 }
gfCNCPoint2[25916] = {X 513.5214, Y 29.5808, Z -3.8333, A 0.000, B 0.000, C 0.000 }
gfCNCPoint2[25917] = {X 513.8068, Y 29.4125, Z -3.8333, A 0.000, B 0.000, C 0.000 }
gfCNCPoint2[25918] = {X 513.8068, Y 27.6757, Z -3.8333, A 0.000, B 0.000, C 0.000 }
gfCNCPoint2[25919] = {X 513.5213, Y 27.5010, Z -3.8333, A 0.000, B 0.000, C 0.000 }
gfCNCPoint2[25920] = {X 513.2409, Y 27.3185, Z -3.8333, A 0.000, B 0.000, C 0.000 }
gfCNCPoint2[25921] = {X 513.2409, Y 29.7568, Z -3.8333, A 0.000, B 0.000, C 0.000 }
gfCNCPoint2[25922] = {X 514.5440, Y 31.7722, Z -3.8333, A 0.000, B 0.000, C 0.000 }
gfCNCPoint2[25923] = {X 515.3545, Y 31.3021, Z -3.8333, A 0.000, B 0.000, C 0.000 }
gfCNCPoint2[25924] = {X 516.2068, Y 30.9126, Z -3.8333, A 0.000, B 0.000, C 0.000 }
gfCNCPoint2[25925] = {X 516.2068, Y 26.2046, Z -3.8333, A 0.000, B 0.000, C 0.000 }
gfCNCPoint2[25926] = {X 515.3711, Y 25.8040, Z -3.8333, A 0.000, B 0.000, C 0.000 }
gfCNCPoint2[25927] = {X 514.5776, Y 25.3252, Z -3.8333, A 0.000, B 0.000, C 0.000 }
gfCNCPoint2[25928] = {X 513.5943, Y 24.5702, Z -3.8333, A 0.000, B 0.000, C 0.000 }
gfCNCPoint2[25929] = {X 512.7156, Y 23.6957, Z -3.8333, A 0.000, B 0.000, C 0.000 }
gfCNCPoint2[25930] = {X 511.9558, Y 22.7161, Z -3.8333, A 0.000, B 0.000, C 0.000 }
gfCNCPoint2[25931] = {X 511.3275, Y 21.6474, Z -3.8333, A 0.000, B 0.000, C 0.000 }
gfCNCPoint2[25932] = {X 510.8409, Y 20.5072, Z -3.8333, A 0.000, B 0.000, C 0.000 }
gfCNCPoint2[25933] = {X 510.8408, Y 36.2351, Z -3.8333, A 0.000, B 0.000, C 0.000 }
gfCNCPoint2[25934] = {X 511.4998, Y 34.9199, Z -3.8333, A 0.000, B 0.000, C 0.000 }
gfCNCPoint2[25935] = {X 512.3503, Y 33.7198, Z -3.8333, A 0.000, B 0.000, C 0.000 }
gfCNCPoint2[25936] = {X 513.3729, Y 32.6624, Z -3.8333, A 0.000, B 0.000, C 0.000 }
gfCNCPoint2[25937] = {X 514.5440, Y 31.7722, Z -3.8333, A 0.000, B 0.000, C 0.000 }
gfCNCPoint2[25938] = {X 515.8471, Y 33.7876, Z -3.8333, A 0.000, B 0.000, C 0.000 }
gfCNCPoint2[25939] = {X 516.7436, Y 33.2937, Z -3.8333, A 0.000, B 0.000, C 0.000 }
gfCNCPoint2[25940] = {X 517.7006, Y 32.9303, Z -3.8333, A 0.000, B 0.000, C 0.000 }
gfCNCPoint2[25941] = {X 518.6990, Y 32.7048, Z -3.8333, A 0.000, B 0.000, C 0.000 }
gfCNCPoint2[25942] = {X 518.6299, Y 32.1290, Z -3.8333, A 0.000, B 0.000, C 0.000 }
gfCNCPoint2[25943] = {X 518.6068, Y 31.5494, Z -3.8333, A 0.000, B 0.000, C 0.000 }
gfCNCPoint2[25944] = {X 518.6068, Y 24.5714, Z -3.8333, A 0.000, B 0.000, C 0.000 }
gfCNCPoint2[25945] = {X 518.6080, Y 24.4373, Z -3.8333, A 0.000, B 0.000, C 0.000 }
gfCNCPoint2[25946] = {X 517.3911, Y 24.0939, Z -3.8333, A 0.000, B 0.000, C 0.000 }
gfCNCPoint2[25947] = {X 516.2519, Y 23.5452, Z -3.8333, A 0.000, B 0.000, C 0.000 }
gfCNCPoint2[25948] = {X 515.2249, Y 22.8075, Z -3.8333, A 0.000, B 0.000, C 0.000 }
gfCNCPoint2[25949] = {X 514.3410, Y 21.9033, Z -3.8333, A 0.000, B 0.000, C 0.000 }
gfCNCPoint2[25950] = {X 513.6269, Y 20.8598, Z -3.8333, A 0.000, B 0.000, C 0.000 }
gfCNCPoint2[25951] = {X 513.1041, Y 19.7085, Z -3.8333, A 0.000, B 0.000, C 0.000 }
gfCNCPoint2[25952] = {X 512.7936, Y 18.5147, Z -3.8333, A 0.000, B 0.000, C 0.000 }
gfCNCPoint2[25953] = {X 512.6891, Y 17.2857, Z -3.8333, A 0.000, B 0.000, C 0.000 }
gfCNCPoint2[25954] = {X 512.6891, Y 10.3077, Z -3.8333, A 0.000, B 0.000, C 0.000 }
gfCNCPoint2[25955] = {X 512.7002, Y 9.9057, Z -3.8333, A 0.000, B 0.000, C 0.000 }
gfCNCPoint2[25956] = {X 512.7335, Y 9.5050, Z -3.8333, A 0.000, B 0.000, C 0.000 }
gfCNCPoint2[25957] = {X 509.4589, Y 9.5050, Z -3.8333, A 0.000, B 0.000, C 0.000 }
gfCNCPoint2[25958] = {X 509.7405, Y 10.3721, Z -3.8333, A 0.000, B 0.000, C 0.000 }
gfCNCPoint2[25959] = {X 509.9113, Y 11.2677, Z -3.8333, A 0.000, B 0.000, C 0.000 }
gfCNCPoint2[25960] = {X 509.9685, Y 12.1776, Z -3.8333, A 0.000, B 0.000, C 0.000 }
gfCNCPoint2[25961] = {X 509.9682, Y 13.0462, Z -3.8333, A 0.000, B 0.000, C 0.000 }
gfCNCPoint2[25962] = {X 509.8611, Y 14.2237, Z -3.8333, A 0.000, B 0.000, C 0.000 }
gfCNCPoint2[25963] = {X 509.5649, Y 15.3683, Z -3.8333, A 0.000, B 0.000, C 0.000 }
gfCNCPoint2[25964] = {X 509.0873, Y 16.4499, Z -3.8333, A 0.000, B 0.000, C 0.000 }
gfCNCPoint2[25965] = {X 508.4409, Y 17.4399, Z -3.8333, A 0.000, B 0.000, C 0.000 }
gfCNCPoint2[25966] = {X 508.4408, Y 39.7468, Z -3.8333, A 0.000, B 0.000, C 0.000 }
gfCNCPoint2[25967] = {X 509.0891, Y 40.7402, Z -3.8333, A 0.000, B 0.000, C 0.000 }
gfCNCPoint2[25968] = {X 509.5674, Y 41.8256, Z -3.8333, A 0.000, B 0.000, C 0.000 }
gfCNCPoint2[25969] = {X 509.8631, Y 42.9743, Z -3.8333, A 0.000, B 0.000, C 0.000 }
gfCNCPoint2[25970] = {X 509.9683, Y 44.1558, Z -3.8333, A 0.000, B 0.000, C 0.000 }
gfCNCPoint2[25971] = {X 509.9685, Y 45.0000, Z -3.8333, A 0.000, B 0.000, C 0.000 }
gfCNCPoint2[25972] = {X 509.8909, Y 46.0603, Z -3.8333, A 0.000, B 0.000, C 0.000 }
gfCNCPoint2[25973] = {X 509.6596, Y 47.0980, Z -3.8333, A 0.000, B 0.000, C 0.000 }
gfCNCPoint2[25974] = {X 509.2797, Y 48.0910, Z -3.8333, A 0.000, B 0.000, C 0.000 }
gfCNCPoint2[25975] = {X 508.7593, Y 49.0180, Z -3.8333, A 0.000, B 0.000, C 0.000 }
gfCNCPoint2[25976] = {X 508.0200, Y 49.9571, Z -3.8333, A 0.000, B 0.000, C 0.000 }
gfCNCPoint2[25977] = {X 507.1371, Y 50.7626, Z -3.8333, A 0.000, B 0.000, C 0.000 }
gfCNCPoint2[25978] = {X 506.1343, Y 51.4129, Z -3.8333, A 0.000, B 0.000, C 0.000 }
gfCNCPoint2[25979] = {X 505.0386, Y 51.8902, Z -3.8333, A 0.000, B 0.000, C 0.000 }
gfCNCPoint2[25980] = {X 503.8796, Y 52.1819, Z -3.8333, A 0.000, B 0.000, C 0.000 }
gfCNCPoint2[25981] = {X 502.6885, Y 52.2800, Z -3.8333, A 0.000, B 0.000, C 0.000 }
gfCNCPoint2[25982] = {X 496.2450, Y 52.2800, Z -3.8333, A 0.000, B 0.000, C 0.000 }
gfCNCPoint2[25983] = {X 495.0845, Y 52.1869, Z -3.8333, A 0.000, B 0.000, C 0.000 }
gfCNCPoint2[25984] = {X 493.9538, Y 51.9100, Z -3.8333, A 0.000, B 0.000, C 0.000 }
gfCNCPoint2[25985] = {X 492.8816, Y 51.4564, Z -3.8333, A 0.000, B 0.000, C 0.000 }
gfCNCPoint2[25986] = {X 491.8954, Y 50.8377, Z -3.8333, A 0.000, B 0.000, C 0.000 }
gfCNCPoint2[25987] = {X 491.0204, Y 50.0697, Z -3.8333, A 0.000, B 0.000, C 0.000 }
gfCNCPoint2[25988] = {X 490.2980, Y 49.1989, Z -3.8333, A 0.000, B 0.000, C 0.000 }
gfCNCPoint2[25989] = {X 489.7192, Y 48.2267, Z -3.8333, A 0.000, B 0.000, C 0.000 }
gfCNCPoint2[25990] = {X 489.2980, Y 47.1766, Z -3.8333, A 0.000, B 0.000, C 0.000 }
gfCNCPoint2[25991] = {X 488.8769, Y 48.2267, Z -3.8333, A 0.000, B 0.000, C 0.000 }
gfCNCPoint2[25992] = {X 488.2981, Y 49.1989, Z -3.8333, A 0.000, B 0.000, C 0.000 }
gfCNCPoint2[25993] = {X 487.5756, Y 50.0697, Z -3.8333, A 0.000, B 0.000, C 0.000 }
gfCNCPoint2[25994] = {X 486.8824, Y 50.6978, Z -3.8333, A 0.000, B 0.000, C 0.000 }
gfCNCPoint2[25995] = {X 486.1145, Y 51.2318, Z -3.8333, A 0.000, B 0.000, C 0.000 }
gfCNCPoint2[25996] = {X 485.2843, Y 51.6629, Z -3.8333, A 0.000, B 0.000, C 0.000 }
gfCNCPoint2[25997] = {X 486.0586, Y 53.1385, Z -3.8333, A 0.000, B 0.000, C 0.000 }
gfCNCPoint2[25998] = {X 486.6224, Y 54.7067, Z -3.8333, A 0.000, B 0.000, C 0.000 }
gfCNCPoint2[25999] = {X 486.9651, Y 56.3375, Z -3.8333, A 0.000, B 0.000, C 0.000 }
gfCNCPoint2[26000] = {X 487.0800, Y 58.0000, Z -3.8333, A 0.000, B 0.000, C 0.000 }
gfCNCPoint2[26001] = {X 487.0796, Y 59.0339, Z -3.8333, A 0.000, B 0.000, C 0.000 }
gfCNCPoint2[26002] = {X 486.9596, Y 60.6352, Z -3.8333, A 0.000, B 0.000, C 0.000 }
gfCNCPoint2[26003] = {X 486.6283, Y 62.2065, Z -3.8333, A 0.000, B 0.000, C 0.000 }
gfCNCPoint2[26004] = {X 486.0915, Y 63.7200, Z -3.8333, A 0.000, B 0.000, C 0.000 }
gfCNCPoint2[26005] = {X 485.3587, Y 65.1489, Z -3.8333, A 0.000, B 0.000, C 0.000 }
gfCNCPoint2[26006] = {X 484.4428, Y 66.4680, Z -3.8333, A 0.000, B 0.000, C 0.000 }
gfCNCPoint2[26007] = {X 483.3600, Y 67.6539, Z -3.8333, A 0.000, B 0.000, C 0.000 }
gfCNCPoint2[26008] = {X 483.3603, Y 88.3507, Z -3.8333, A 0.000, B 0.000, C 0.000 }
gfCNCPoint2[26009] = {X 484.3103, Y 89.3714, Z -3.8333, A 0.000, B 0.000, C 0.000 }
gfCNCPoint2[26010] = {X 485.1360, Y 90.4950, Z -3.8333, A 0.000, B 0.000, C 0.000 }
gfCNCPoint2[26011] = {X 507.6816, Y 90.4950, Z -3.8333, A 0.000, B 0.000, C 0.000 }
gfCNCPoint2[26012] = {X 507.6816, Y 92.8950, Z -3.8333, A 0.000, B 0.000, C 0.000 }
gfCNCPoint2[26013] = {X 592.8965, Y 92.8950, Z -3.8333, A 0.000, B 0.000, C 0.000 }
gfCNCPoint2[26014] = {X 592.8965, Y 56.5812, Z -3.8333, A 0.000, B 0.000, C 0.000 }
gfCNCPoint2[26015] = {X 591.4810, Y 56.4128, Z -3.8333, A 0.000, B 0.000, C 0.000 }
gfCNCPoint2[26016] = {X 590.0968, Y 56.0720, Z -3.8333, A 0.000, B 0.000, C 0.000 }
gfCNCPoint2[26017] = {X 588.7648, Y 55.5641, Z -3.8333, A 0.000, B 0.000, C 0.000 }
gfCNCPoint2[26018] = {X 587.5052, Y 54.8965, Z -3.8333, A 0.000, B 0.000, C 0.000 }
gfCNCPoint2[26019] = {X 586.9690, Y 55.2051, Z -3.8333, A 0.000, B 0.000, C 0.000 }
gfCNCPoint2[26020] = {X 586.4171, Y 55.4846, Z -3.8333, A 0.000, B 0.000, C 0.000 }
gfCNCPoint2[26021] = {X 584.8782, Y 56.0830, Z -3.8333, A 0.000, B 0.000, C 0.000 }
gfCNCPoint2[26022] = {X 583.2699, Y 56.4570, Z -3.8333, A 0.000, B 0.000, C 0.000 }
gfCNCPoint2[26023] = {X 581.6248, Y 56.5987, Z -3.8333, A 0.000, B 0.000, C 0.000 }
gfCNCPoint2[26024] = {X 579.9763, Y 56.5055, Z -3.8333, A 0.000, B 0.000, C 0.000 }
gfCNCPoint2[26025] = {X 578.3577, Y 56.1792, Z -3.8333, A 0.000, B 0.000, C 0.000 }
gfCNCPoint2[26026] = {X 576.8018, Y 55.6263, Z -3.8333, A 0.000, B 0.000, C 0.000 }
gfCNCPoint2[26027] = {X 575.3401, Y 54.8581, Z -3.8333, A 0.000, B 0.000, C 0.000 }
gfCNCPoint2[26028] = {X 573.9176, Y 55.6091, Z -3.8333, A 0.000, B 0.000, C 0.000 }
gfCNCPoint2[26029] = {X 572.4049, Y 56.1560, Z -3.8333, A 0.000, B 0.000, C 0.000 }
gfCNCPoint2[26030] = {X 570.8311, Y 56.4885, Z -3.8333, A 0.000, B 0.000, C 0.000 }
gfCNCPoint2[26031] = {X 569.2264, Y 56.6000, Z -3.8333, A 0.000, B 0.000, C 0.000 }
gfCNCPoint2[26032] = {X 562.4443, Y 56.6000, Z -3.8333, A 0.000, B 0.000, C 0.000 }
gfCNCPoint2[26033] = {X 560.8792, Y 56.4939, Z -3.8333, A 0.000, B 0.000, C 0.000 }
gfCNCPoint2[26034] = {X 559.3428, Y 56.1777, Z -3.8333, A 0.000, B 0.000, C 0.000 }
gfCNCPoint2[26035] = {X 557.8631, Y 55.6570, Z -3.8333, A 0.000, B 0.000, C 0.000 }
gfCNCPoint2[26036] = {X 556.4672, Y 54.9415, Z -3.8333, A 0.000, B 0.000, C 0.000 }
gfCNCPoint2[26037] = {X 555.1805, Y 54.0442, Z -3.8333, A 0.000, B 0.000, C 0.000 }
gfCNCPoint2[26038] = {X 554.0267, Y 52.9815, Z -3.8333, A 0.000, B 0.000, C 0.000 }
gfCNCPoint2[26039] = {X 553.0268, Y 51.7728, Z -3.8333, A 0.000, B 0.000, C 0.000 }
gfCNCPoint2[26040] = {X 552.1992, Y 50.4403, Z -3.8333, A 0.000, B 0.000, C 0.000 }
gfCNCPoint2[26041] = {X 551.5588, Y 49.0083, Z -3.8333, A 0.000, B 0.000, C 0.000 }
gfCNCPoint2[26042] = {X 551.1637, Y 47.7034, Z -3.8333, A 0.000, B 0.000, C 0.000 }
gfCNCPoint2[26043] = {X 550.9244, Y 46.3611, Z -3.8333, A 0.000, B 0.000, C 0.000 }
gfCNCPoint2[26044] = {X 550.8443, Y 45.0000, Z -3.8333, A 0.000, B 0.000, C 0.000 }
gfCNCPoint2[26045] = {X 550.8444, Y 44.0325, Z -3.8333, A 0.000, B 0.000, C 0.000 }
gfCNCPoint2[26046] = {X 550.9590, Y 42.4536, Z -3.8333, A 0.000, B 0.000, C 0.000 }
gfCNCPoint2[26047] = {X 551.2869, Y 40.9048, Z -3.8333, A 0.000, B 0.000, C 0.000 }
gfCNCPoint2[26048] = {X 551.8220, Y 39.4149, Z -3.8333, A 0.000, B 0.000, C 0.000 }
gfCNCPoint2[26049] = {X 549.6237, Y 38.4518, Z -3.8333, A 0.000, B 0.000, C 0.000 }
gfCNCPoint2[26050] = {X 549.7926, Y 38.0812, Z -3.8333, A 0.000, B 0.000, C 0.000 }
gfCNCPoint2[26051] = {X 549.9721, Y 37.7155, Z -3.8333, A 0.000, B 0.000, C 0.000 }
gfCNCPoint2[26052] = {X 549.9721, Y 16.9505, Z -3.8333, A 0.000, B 0.000, C 0.000 }
gfCNCPoint2[26053] = {X 549.8029, Y 17.1990, Z -3.8333, A 0.000, B 0.000, C 0.000 }
gfCNCPoint2[26054] = {X 549.6235, Y 17.4403, Z -3.8333, A 0.000, B 0.000, C 0.000 }
gfCNCPoint2[26055] = {X 549.6237, Y 38.4518, Z -3.8333, A 0.000, B 0.000, C 0.000 }
gfCNCPoint2[26056] = {X 551.8220, Y 39.4149, Z -3.8333, A 0.000, B 0.000, C 0.000 }
gfCNCPoint2[26057] = {X 552.0826, Y 38.8602, Z -3.8333, A 0.000, B 0.000, C 0.000 }
gfCNCPoint2[26058] = {X 552.3721, Y 38.3200, Z -3.8333, A 0.000, B 0.000, C 0.000 }
gfCNCPoint2[26059] = {X 552.3721, Y 11.6882, Z -3.8333, A 0.000, B 0.000, C 0.000 }
gfCNCPoint2[26060] = {X 551.6706, Y 10.2339, Z -3.8333, A 0.000, B 0.000, C 0.000 }
gfCNCPoint2[26061] = {X 551.1779, Y 8.6962, Z -3.8333, A 0.000, B 0.000, C 0.000 }
gfCNCPoint2[26062] = {X 550.9035, Y 7.1050, Z -3.8333, A 0.000, B 0.000, C 0.000 }
gfCNCPoint2[26063] = {X 524.2928, Y 7.1050, Z -3.8333, A 0.000, B 0.000, C 0.000 }
gfCNCPoint2[26064] = {X 524.3787, Y 7.2066, Z -3.8333, A 0.000, B 0.000, C 0.000 }
gfCNCPoint2[26065] = {X 524.4618, Y 7.3104, Z -3.8333, A 0.000, B 0.000, C 0.000 }
gfCNCPoint2[26066] = {X 543.7426, Y 7.3109, Z -3.8333, A 0.000, B 0.000, C 0.000 }
gfCNCPoint2[26067] = {X 544.7119, Y 7.3830, Z -3.8333, A 0.000, B 0.000, C 0.000 }
gfCNCPoint2[26068] = {X 545.6476, Y 7.6456, Z -3.8333, A 0.000, B 0.000, C 0.000 }
gfCNCPoint2[26069] = {X 546.5129, Y 8.0882, Z -3.8333, A 0.000, B 0.000, C 0.000 }
gfCNCPoint2[26070] = {X 547.2734, Y 8.6934, Z -3.8333, A 0.000, B 0.000, C 0.000 }
gfCNCPoint2[26071] = {X 547.8990, Y 9.4372, Z -3.8333, A 0.000, B 0.000, C 0.000 }
gfCNCPoint2[26072] = {X 548.3650, Y 10.2901, Z -3.8333, A 0.000, B 0.000, C 0.000 }
gfCNCPoint2[26073] = {X 548.6530, Y 11.2183, Z -3.8333, A 0.000, B 0.000, C 0.000 }
gfCNCPoint2[26074] = {X 548.7514, Y 12.1852, Z -3.8333, A 0.000, B 0.000, C 0.000 }
gfCNCPoint2[26075] = {X 548.7512, Y 13.0283, Z -3.8333, A 0.000, B 0.000, C 0.000 }
gfCNCPoint2[26076] = {X 548.6549, Y 13.9440, Z -3.8333, A 0.000, B 0.000, C 0.000 }
gfCNCPoint2[26077] = {X 548.3883, Y 14.8253, Z -3.8333, A 0.000, B 0.000, C 0.000 }
gfCNCPoint2[26078] = {X 547.9609, Y 15.6409, Z -3.8333, A 0.000, B 0.000, C 0.000 }
gfCNCPoint2[26079] = {X 547.6183, Y 16.1045, Z -3.8333, A 0.000, B 0.000, C 0.000 }
gfCNCPoint2[26080] = {X 547.2235, Y 16.5246, Z -3.8333, A 0.000, B 0.000, C 0.000 }
gfCNCPoint2[26081] = {X 547.2237, Y 40.6625, Z -3.8333, A 0.000, B 0.000, C 0.000 }
gfCNCPoint2[26082] = {X 547.8652, Y 41.4045, Z -3.8333, A 0.000, B 0.000, C 0.000 }
gfCNCPoint2[26083] = {X 548.3453, Y 42.2597, Z -3.8333, A 0.000, B 0.000, C 0.000 }
gfCNCPoint2[26084] = {X 548.6447, Y 43.1937, Z -3.8333, A 0.000, B 0.000, C 0.000 }
gfCNCPoint2[26085] = {X 548.7513, Y 44.1687, Z -3.8333, A 0.000, B 0.000, C 0.000 }
gfCNCPoint2[26086] = {X 548.7514, Y 45.0016, Z -3.8333, A 0.000, B 0.000, C 0.000 }
gfCNCPoint2[26087] = {X 548.6696, Y 45.8829, Z -3.8333, A 0.000, B 0.000, C 0.000 }
gfCNCPoint2[26088] = {X 548.4301, Y 46.7349, Z -3.8333, A 0.000, B 0.000, C 0.000 }
gfCNCPoint2[26089] = {X 548.0408, Y 47.5298, Z -3.8333, A 0.000, B 0.000, C 0.000 }
gfCNCPoint2[26090] = {X 547.5145, Y 48.2414, Z -3.8333, A 0.000, B 0.000, C 0.000 }
gfCNCPoint2[26091] = {X 546.7288, Y 48.9509, Z -3.8333, A 0.000, B 0.000, C 0.000 }
gfCNCPoint2[26092] = {X 545.8088, Y 49.4746, Z -3.8333, A 0.000, B 0.000, C 0.000 }
gfCNCPoint2[26093] = {X 544.7976, Y 49.7877, Z -3.8333, A 0.000, B 0.000, C 0.000 }
gfCNCPoint2[26094] = {X 543.7426, Y 49.8756, Z -3.8333, A 0.000, B 0.000, C 0.000 }
gfCNCPoint2[26095] = {X 524.3234, Y 49.8761, Z -3.8333, A 0.000, B 0.000, C 0.000 }
gfCNCPoint2[26096] = {X 523.7106, Y 50.5150, Z -3.8333, A 0.000, B 0.000, C 0.000 }
gfCNCPoint2[26097] = {X 522.9954, Y 51.0367, Z -3.8333, A 0.000, B 0.000, C 0.000 }
gfCNCPoint2[26098] = {X 522.1999, Y 51.4253, Z -3.8333, A 0.000, B 0.000, C 0.000 }
gfCNCPoint2[26099] = {X 521.3487, Y 51.6686, Z -3.8333, A 0.000, B 0.000, C 0.000 }
gfCNCPoint2[26100] = {X 520.4681, Y 51.7591, Z -3.8333, A 0.000, B 0.000, C 0.000 }
gfCNCPoint2[26101] = {X 519.7998, Y 51.7591, Z -3.8333, A 0.000, B 0.000, C 0.000 }
gfCNCPoint2[26102] = {X 518.8477, Y 51.6654, Z -3.8333, A 0.000, B 0.000, C 0.000 }
gfCNCPoint2[26103] = {X 517.9323, Y 51.3877, Z -3.8333, A 0.000, B 0.000, C 0.000 }
gfCNCPoint2[26104] = {X 517.0886, Y 50.9367, Z -3.8333, A 0.000, B 0.000, C 0.000 }
gfCNCPoint2[26105] = {X 516.3491, Y 50.3298, Z -3.8333, A 0.000, B 0.000, C 0.000 }
gfCNCPoint2[26106] = {X 515.7422, Y 49.5903, Z -3.8333, A 0.000, B 0.000, C 0.000 }
gfCNCPoint2[26107] = {X 515.2912, Y 48.7466, Z -3.8333, A 0.000, B 0.000, C 0.000 }
gfCNCPoint2[26108] = {X 515.0135, Y 47.8312, Z -3.8333, A 0.000, B 0.000, C 0.000 }
gfCNCPoint2[26109] = {X 514.9198, Y 46.8791, Z -3.8333, A 0.000, B 0.000, C 0.000 }
gfCNCPoint2[26110] = {X 514.9198, Y 39.9011, Z -3.8333, A 0.000, B 0.000, C 0.000 }
gfCNCPoint2[26111] = {X 515.0197, Y 38.9186, Z -3.8333, A 0.000, B 0.000, C 0.000 }
gfCNCPoint2[26112] = {X 515.3154, Y 37.9764, Z -3.8333, A 0.000, B 0.000, C 0.000 }
gfCNCPoint2[26113] = {X 515.7947, Y 37.1129, Z -3.8333, A 0.000, B 0.000, C 0.000 }
gfCNCPoint2[26114] = {X 516.4381, Y 36.3637, Z -3.8333, A 0.000, B 0.000, C 0.000 }
gfCNCPoint2[26115] = {X 517.2191, Y 35.7593, Z -3.8333, A 0.000, B 0.000, C 0.000 }
gfCNCPoint2[26116] = {X 518.1058, Y 35.3245, Z -3.8333, A 0.000, B 0.000, C 0.000 }
gfCNCPoint2[26117] = {X 519.0619, Y 35.0772, Z -3.8333, A 0.000, B 0.000, C 0.000 }
gfCNCPoint2[26118] = {X 519.4084, Y 35.0368, Z -3.8333, A 0.000, B 0.000, C 0.000 }
gfCNCPoint2[26119] = {X 519.7568, Y 35.0213, Z -3.8333, A 0.000, B 0.000, C 0.000 }
gfCNCPoint2[26120] = {X 520.5345, Y 35.0215, Z -3.8333, A 0.000, B 0.000, C 0.000 }
gfCNCPoint2[26121] = {X 521.4085, Y 35.1125, Z -3.8333, A 0.000, B 0.000, C 0.000 }
gfCNCPoint2[26122] = {X 522.2520, Y 35.3588, Z -3.8333, A 0.000, B 0.000, C 0.000 }
gfCNCPoint2[26123] = {X 523.0377, Y 35.7524, Z -3.8333, A 0.000, B 0.000, C 0.000 }
gfCNCPoint2[26124] = {X 523.7401, Y 36.2804, Z -3.8333, A 0.000, B 0.000, C 0.000 }
gfCNCPoint2[26125] = {X 524.3363, Y 36.9259, Z -3.8333, A 0.000, B 0.000, C 0.000 }
gfCNCPoint2[26126] = {X 534.0719, Y 36.9264, Z -3.8333, A 0.000, B 0.000, C 0.000 }
gfCNCPoint2[26127] = {X 534.0719, Y 34.5252, Z -3.8333, A 0.000, B 0.000, C 0.000 }
gfCNCPoint2[26128] = {X 530.3964, Y 34.5248, Z -3.8333, A 0.000, B 0.000, C 0.000 }
gfCNCPoint2[26129] = {X 529.7965, Y 35.1735, Z -3.8333, A 0.000, B 0.000, C 0.000 }
gfCNCPoint2[26130] = {X 529.0895, Y 35.7034, Z -3.8333, A 0.000, B 0.000, C 0.000 }
gfCNCPoint2[26131] = {X 528.2985, Y 36.0971, Z -3.8333, A 0.000, B 0.000, C 0.000 }
gfCNCPoint2[26132] = {X 527.4495, Y 36.3417, Z -3.8333, A 0.000, B 0.000, C 0.000 }
gfCNCPoint2[26133] = {X 526.5703, Y 36.4293, Z -3.8333, A 0.000, B 0.000, C 0.000 }
gfCNCPoint2[26134] = {X 525.8868, Y 36.4294, Z -3.8333, A 0.000, B 0.000, C 0.000 }
gfCNCPoint2[26135] = {X 524.9094, Y 36.3306, Z -3.8333, A 0.000, B 0.000, C 0.000 }
gfCNCPoint2[26136] = {X 523.9717, Y 36.0380, Z -3.8333, A 0.000, B 0.000, C 0.000 }
gfCNCPoint2[26137] = {X 523.1116, Y 35.5636, Z -3.8333, A 0.000, B 0.000, C 0.000 }
gfCNCPoint2[26138] = {X 522.3639, Y 34.9265, Z -3.8333, A 0.000, B 0.000, C 0.000 }
gfCNCPoint2[26139] = {X 521.7590, Y 34.1525, Z -3.8333, A 0.000, B 0.000, C 0.000 }
gfCNCPoint2[26140] = {X 521.3213, Y 33.2731, Z -3.8333, A 0.000, B 0.000, C 0.000 }
gfCNCPoint2[26141] = {X 521.0686, Y 32.3239, Z -3.8333, A 0.000, B 0.000, C 0.000 }
gfCNCPoint2[26142] = {X 521.0222, Y 31.9379, Z -3.8333, A 0.000, B 0.000, C 0.000 }
gfCNCPoint2[26143] = {X 521.0068, Y 31.5494, Z -3.8333, A 0.000, B 0.000, C 0.000 }
gfCNCPoint2[26144] = {X 521.0076, Y 24.4815, Z -3.8333, A 0.000, B 0.000, C 0.000 }
gfCNCPoint2[26145] = {X 521.0984, Y 23.6300, Z -3.8333, A 0.000, B 0.000, C 0.000 }
gfCNCPoint2[26146] = {X 521.3368, Y 22.8074, Z -3.8333, A 0.000, B 0.000, C 0.000 }
gfCNCPoint2[26147] = {X 521.7152, Y 22.0391, Z -3.8333, A 0.000, B 0.000, C 0.000 }
gfCNCPoint2[26148] = {X 521.1864, Y 22.1316, Z -3.8333, A 0.000, B 0.000, C 0.000 }
gfCNCPoint2[26149] = {X 520.6505, Y 22.1656, Z -3.8333, A 0.000, B 0.000, C 0.000 }
gfCNCPoint2[26150] = {X 519.9691, Y 22.1657, Z -3.8333, A 0.000, B 0.000, C 0.000 }
gfCNCPoint2[26151] = {X 519.5109, Y 22.1442, Z -3.8333, A 0.000, B 0.000, C 0.000 }
gfCNCPoint2[26152] = {X 519.0567, Y 22.0797, Z -3.8333, A 0.000, B 0.000, C 0.000 }
gfCNCPoint2[26153] = {X 518.1336, Y 21.8074, Z -3.8333, A 0.000, B 0.000, C 0.000 }
gfCNCPoint2[26154] = {X 517.2820, Y 21.3592, Z -3.8333, A 0.000, B 0.000, C 0.000 }
gfCNCPoint2[26155] = {X 516.5348, Y 20.7527, Z -3.8333, A 0.000, B 0.000, C 0.000 }
gfCNCPoint2[26156] = {X 515.9212, Y 20.0113, Z -3.8333, A 0.000, B 0.000, C 0.000 }
gfCNCPoint2[26157] = {X 515.4650, Y 19.1639, Z -3.8333, A 0.000, B 0.000, C 0.000 }
gfCNCPoint2[26158] = {X 515.1840, Y 18.2434, Z -3.8333, A 0.000, B 0.000, C 0.000 }
gfCNCPoint2[26159] = {X 515.0891, Y 17.2857, Z -3.8333, A 0.000, B 0.000, C 0.000 }
gfCNCPoint2[26160] = {X 515.0891, Y 10.3077, Z -3.8333, A 0.000, B 0.000, C 0.000 }
gfCNCPoint2[26161] = {X 515.0965, Y 10.0382, Z -3.8333, A 0.000, B 0.000, C 0.000 }
gfCNCPoint2[26162] = {X 515.1189, Y 9.7696, Z -3.8333, A 0.000, B 0.000, C 0.000 }
gfCNCPoint2[26163] = {X 515.3251, Y 8.8084, Z -3.8333, A 0.000, B 0.000, C 0.000 }
gfCNCPoint2[26164] = {X 515.7199, Y 7.9080, Z -3.8333, A 0.000, B 0.000, C 0.000 }
gfCNCPoint2[26165] = {X 516.2871, Y 7.1050, Z -3.8333, A 0.000, B 0.000, C 0.000 }
gfCNCPoint2[26166] = {X 516.6493, Y 7.4200, Z -3.8333, A 0.000, B 0.000, C 0.000 }
gfCNCPoint2[26167] = {X 517.3373, Y 6.7816, Z -3.8333, A 0.000, B 0.000, C 0.000 }
gfCNCPoint2[26168] = {X 518.1451, Y 6.3036, Z -3.8333, A 0.000, B 0.000, C 0.000 }
gfCNCPoint2[26169] = {X 519.0359, Y 6.0078, Z -3.8333, A 0.000, B 0.000, C 0.000 }
gfCNCPoint2[26170] = {X 519.9692, Y 5.9077, Z -3.8333, A 0.000, B 0.000, C 0.000 }
gfCNCPoint2[26171] = {X 520.6509, Y 5.9079, Z -3.8333, A 0.000, B 0.000, C 0.000 }
gfCNCPoint2[26172] = {X 521.4834, Y 5.9951, Z -3.8333, A 0.000, B 0.000, C 0.000 }
gfCNCPoint2[26173] = {X 522.2843, Y 6.2384, Z -3.8333, A 0.000, B 0.000, C 0.000 }
gfCNCPoint2[26174] = {X 523.0246, Y 6.6289, Z -3.8333, A 0.000, B 0.000, C 0.000 }
gfCNCPoint2[26175] = {X 523.6776, Y 7.1526, Z -3.8333, A 0.000, B 0.000, C 0.000 }
gfCNCPoint2[26176] = {X 524.2196, Y 7.7904, Z -3.8333, A 0.000, B 0.000, C 0.000 }
gfCNCPoint2[26177] = {X 543.7489, Y 7.7909, Z -3.8333, A 0.000, B 0.000, C 0.000 }
gfCNCPoint2[26178] = {X 544.7470, Y 7.8782, Z -3.8333, A 0.000, B 0.000, C 0.000 }
gfCNCPoint2[26179] = {X 545.6996, Y 8.1888, Z -3.8333, A 0.000, B 0.000, C 0.000 }
gfCNCPoint2[26180] = {X 546.5573, Y 8.7067, Z -3.8333, A 0.000, B 0.000, C 0.000 }
gfCNCPoint2[26181] = {X 547.2758, Y 9.4050, Z -3.8333, A 0.000, B 0.000, C 0.000 }
gfCNCPoint2[26182] = {X 547.8180, Y 10.2476, Z -3.8333, A 0.000, B 0.000, C 0.000 }
gfCNCPoint2[26183] = {X 548.1556, Y 11.1909, Z -3.8333, A 0.000, B 0.000, C 0.000 }
gfCNCPoint2[26184] = {X 548.2714, Y 12.1861, Z -3.8333, A 0.000, B 0.000, C 0.000 }
gfCNCPoint2[26185] = {X 548.2712, Y 13.0233, Z -3.8333, A 0.000, B 0.000, C 0.000 }
gfCNCPoint2[26186] = {X 548.1628, Y 13.9495, Z -3.8333, A 0.000, B 0.000, C 0.000 }
gfCNCPoint2[26187] = {X 547.8618, Y 14.8320, Z -3.8333, A 0.000, B 0.000, C 0.000 }
gfCNCPoint2[26188] = {X 547.3815, Y 15.6313, Z -3.8333, A 0.000, B 0.000, C 0.000 }
gfCNCPoint2[26189] = {X 546.7435, Y 16.3114, Z -3.8333, A 0.000, B 0.000, C 0.000 }
gfCNCPoint2[26190] = {X 546.7437, Y 40.8757, Z -3.8333, A 0.000, B 0.000, C 0.000 }
gfCNCPoint2[26191] = {X 547.3884, Y 41.5648, Z -3.8333, A 0.000, B 0.000, C 0.000 }
gfCNCPoint2[26192] = {X 547.8713, Y 42.3756, Z -3.8333, A 0.000, B 0.000, C 0.000 }
gfCNCPoint2[26193] = {X 548.1703, Y 43.2707, Z -3.8333, A 0.000, B 0.000, C 0.000 }
gfCNCPoint2[26194] = {X 548.2714, Y 44.2089, Z -3.8333, A 0.000, B 0.000, C 0.000 }
gfCNCPoint2[26195] = {X 548.2714, Y 45.0007, Z -3.8333, A 0.000, B 0.000, C 0.000 }
gfCNCPoint2[26196] = {X 548.1557, Y 45.9959, Z -3.8333, A 0.000, B 0.000, C 0.000 }
gfCNCPoint2[26197] = {X 547.8180, Y 46.9392, Z -3.8333, A 0.000, B 0.000, C 0.000 }
gfCNCPoint2[26198] = {X 547.2758, Y 47.7818, Z -3.8333, A 0.000, B 0.000, C 0.000 }
gfCNCPoint2[26199] = {X 546.5573, Y 48.4800, Z -3.8333, A 0.000, B 0.000, C 0.000 }
gfCNCPoint2[26200] = {X 545.6996, Y 48.9978, Z -3.8333, A 0.000, B 0.000, C 0.000 }
gfCNCPoint2[26201] = {X 544.7470, Y 49.3084, Z -3.8333, A 0.000, B 0.000, C 0.000 }
gfCNCPoint2[26202] = {X 543.7489, Y 49.3956, Z -3.8333, A 0.000, B 0.000, C 0.000 }
gfCNCPoint2[26203] = {X 524.0861, Y 49.3961, Z -3.8333, A 0.000, B 0.000, C 0.000 }
gfCNCPoint2[26204] = {X 523.5293, Y 50.0311, Z -3.8333, A 0.000, B 0.000, C 0.000 }
gfCNCPoint2[26205] = {X 522.8650, Y 50.5525, Z -3.8333, A 0.000, B 0.000, C 0.000 }
gfCNCPoint2[26206] = {X 522.1158, Y 50.9424, Z -3.8333, A 0.000, B 0.000, C 0.000 }
gfCNCPoint2[26207] = {X 521.3076, Y 51.1874, Z -3.8333, A 0.000, B 0.000, C 0.000 }
gfCNCPoint2[26208] = {X 520.4681, Y 51.2791, Z -3.8333, A 0.000, B 0.000, C 0.000 }
gfCNCPoint2[26209] = {X 519.7998, Y 51.2791, Z -3.8333, A 0.000, B 0.000, C 0.000 }
gfCNCPoint2[26210] = {X 518.8207, Y 51.1688, Z -3.8333, A 0.000, B 0.000, C 0.000 }
gfCNCPoint2[26211] = {X 517.8907, Y 50.8434, Z -3.8333, A 0.000, B 0.000, C 0.000 }
gfCNCPoint2[26212] = {X 517.0564, Y 50.3192, Z -3.8333, A 0.000, B 0.000, C 0.000 }
gfCNCPoint2[26213] = {X 516.3597, Y 49.6225, Z -3.8333, A 0.000, B 0.000, C 0.000 }
gfCNCPoint2[26214] = {X 515.8355, Y 48.7882, Z -3.8333, A 0.000, B 0.000, C 0.000 }
gfCNCPoint2[26215] = {X 515.5101, Y 47.8582, Z -3.8333, A 0.000, B 0.000, C 0.000 }
gfCNCPoint2[26216] = {X 515.3998, Y 46.8791, Z -3.8333, A 0.000, B 0.000, C 0.000 }
gfCNCPoint2[26217] = {X 515.3998, Y 39.9011, Z -3.8333, A 0.000, B 0.000, C 0.000 }
gfCNCPoint2[26218] = {X 515.5101, Y 38.9220, Z -3.8333, A 0.000, B 0.000, C 0.000 }
gfCNCPoint2[26219] = {X 515.8355, Y 37.9920, Z -3.8333, A 0.000, B 0.000, C 0.000 }
gfCNCPoint2[26220] = {X 516.3597, Y 37.1577, Z -3.8333, A 0.000, B 0.000, C 0.000 }
gfCNCPoint2[26221] = {X 517.0565, Y 36.4610, Z -3.8333, A 0.000, B 0.000, C 0.000 }
gfCNCPoint2[26222] = {X 517.8907, Y 35.9368, Z -3.8333, A 0.000, B 0.000, C 0.000 }
gfCNCPoint2[26223] = {X 518.8207, Y 35.6114, Z -3.8333, A 0.000, B 0.000, C 0.000 }
gfCNCPoint2[26224] = {X 519.7998, Y 35.5011, Z -3.8333, A 0.000, B 0.000, C 0.000 }
gfCNCPoint2[26225] = {X 520.5280, Y 35.5015, Z -3.8333, A 0.000, B 0.000, C 0.000 }
gfCNCPoint2[26226] = {X 521.3614, Y 35.5927, Z -3.8333, A 0.000, B 0.000, C 0.000 }
gfCNCPoint2[26227] = {X 522.1625, Y 35.8404, Z -3.8333, A 0.000, B 0.000, C 0.000 }
gfCNCPoint2[26228] = {X 522.9020, Y 36.2355, Z -3.8333, A 0.000, B 0.000, C 0.000 }
gfCNCPoint2[26229] = {X 523.5532, Y 36.7637, Z -3.8333, A 0.000, B 0.000, C 0.000 }
gfCNCPoint2[26230] = {X 524.0923, Y 37.4059, Z -3.8333, A 0.000, B 0.000, C 0.000 }
gfCNCPoint2[26231] = {X 534.5519, Y 37.4064, Z -3.8333, A 0.000, B 0.000, C 0.000 }
gfCNCPoint2[26232] = {X 534.5519, Y 34.0452, Z -3.8333, A 0.000, B 0.000, C 0.000 }
gfCNCPoint2[26233] = {X 530.1524, Y 34.0448, Z -3.8333, A 0.000, B 0.000, C 0.000 }
gfCNCPoint2[26234] = {X 529.6047, Y 34.6953, Z -3.8333, A 0.000, B 0.000, C 0.000 }
gfCNCPoint2[26235] = {X 528.9421, Y 35.2283, Z -3.8333, A 0.000, B 0.000, C 0.000 }
gfCNCPoint2[26236] = {X 528.1894, Y 35.6239, Z -3.8333, A 0.000, B 0.000, C 0.000 }
gfCNCPoint2[26237] = {X 527.3746, Y 35.8673, Z -3.8333, A 0.000, B 0.000, C 0.000 }
gfCNCPoint2[26238] = {X 526.5283, Y 35.9495, Z -3.8333, A 0.000, B 0.000, C 0.000 }
gfCNCPoint2[26239] = {X 525.8868, Y 35.9495, Z -3.8333, A 0.000, B 0.000, C 0.000 }
gfCNCPoint2[26240] = {X 524.9077, Y 35.8391, Z -3.8333, A 0.000, B 0.000, C 0.000 }
gfCNCPoint2[26241] = {X 523.9777, Y 35.5137, Z -3.8333, A 0.000, B 0.000, C 0.000 }
gfCNCPoint2[26242] = {X 523.1434, Y 34.9895, Z -3.8333, A 0.000, B 0.000, C 0.000 }
gfCNCPoint2[26243] = {X 522.4467, Y 34.2928, Z -3.8333, A 0.000, B 0.000, C 0.000 }
gfCNCPoint2[26244] = {X 521.9225, Y 33.4585, Z -3.8333, A 0.000, B 0.000, C 0.000 }
gfCNCPoint2[26245] = {X 521.5971, Y 32.5285, Z -3.8333, A 0.000, B 0.000, C 0.000 }
gfCNCPoint2[26246] = {X 521.4868, Y 31.5495, Z -3.8333, A 0.000, B 0.000, C 0.000 }
gfCNCPoint2[26247] = {X 521.4868, Y 24.5714, Z -3.8333, A 0.000, B 0.000, C 0.000 }
gfCNCPoint2[26248] = {X 521.5971, Y 23.5923, Z -3.8333, A 0.000, B 0.000, C 0.000 }
gfCNCPoint2[26249] = {X 521.9225, Y 22.6623, Z -3.8333, A 0.000, B 0.000, C 0.000 }
gfCNCPoint2[26250] = {X 522.4467, Y 21.8281, Z -3.8333, A 0.000, B 0.000, C 0.000 }
gfCNCPoint2[26251] = {X 523.1434, Y 21.1314, Z -3.8333, A 0.000, B 0.000, C 0.000 }
gfCNCPoint2[26252] = {X 523.9777, Y 20.6072, Z -3.8333, A 0.000, B 0.000, C 0.000 }
gfCNCPoint2[26253] = {X 524.9077, Y 20.2817, Z -3.8333, A 0.000, B 0.000, C 0.000 }
gfCNCPoint2[26254] = {X 525.8868, Y 20.1714, Z -3.8333, A 0.000, B 0.000, C 0.000 }
gfCNCPoint2[26255] = {X 526.5702, Y 20.1716, Z -3.8333, A 0.000, B 0.000, C 0.000 }
gfCNCPoint2[26256] = {X 527.4023, Y 20.2591, Z -3.8333, A 0.000, B 0.000, C 0.000 }
gfCNCPoint2[26257] = {X 528.2028, Y 20.5025, Z -3.8333, A 0.000, B 0.000, C 0.000 }
gfCNCPoint2[26258] = {X 528.9428, Y 20.8930, Z -3.8333, A 0.000, B 0.000, C 0.000 }
gfCNCPoint2[26259] = {X 529.5954, Y 21.4165, Z -3.8333, A 0.000, B 0.000, C 0.000 }
gfCNCPoint2[26260] = {X 530.1372, Y 22.0541, Z -3.8333, A 0.000, B 0.000, C 0.000 }
gfCNCPoint2[26261] = {X 534.5519, Y 22.0544, Z -3.8333, A 0.000, B 0.000, C 0.000 }
gfCNCPoint2[26262] = {X 534.5519, Y 19.7816, Z -3.8333, A 0.000, B 0.000, C 0.000 }
gfCNCPoint2[26263] = {X 528.8172, Y 19.7815, Z -3.8333, A 0.000, B 0.000, C 0.000 }
gfCNCPoint2[26264] = {X 528.8172, Y 20.2615, Z -3.8333, A 0.000, B 0.000, C 0.000 }
gfCNCPoint2[26265] = {X 534.0719, Y 20.2616, Z -3.8333, A 0.000, B 0.000, C 0.000 }
gfCNCPoint2[26266] = {X 534.0719, Y 21.5744, Z -3.8333, A 0.000, B 0.000, C 0.000 }
gfCNCPoint2[26267] = {X 530.3795, Y 21.5741, Z -3.8333, A 0.000, B 0.000, C 0.000 }
gfCNCPoint2[26268] = {X 529.6677, Y 20.8352, Z -3.8333, A 0.000, B 0.000, C 0.000 }
gfCNCPoint2[26269] = {X 528.8172, Y 20.2615, Z -3.8333, A 0.000, B 0.000, C 0.000 }
gfCNCPoint2[26270] = {X 528.8172, Y 19.7815, Z -3.8333, A 0.000, B 0.000, C 0.000 }
gfCNCPoint2[26271] = {X 524.2346, Y 19.7813, Z -3.8333, A 0.000, B 0.000, C 0.000 }
gfCNCPoint2[26272] = {X 523.6869, Y 20.4317, Z -3.8333, A 0.000, B 0.000, C 0.000 }
gfCNCPoint2[26273] = {X 523.0244, Y 20.9646, Z -3.8333, A 0.000, B 0.000, C 0.000 }
gfCNCPoint2[26274] = {X 522.2717, Y 21.3602, Z -3.8333, A 0.000, B 0.000, C 0.000 }
gfCNCPoint2[26275] = {X 521.4570, Y 21.6036, Z -3.8333, A 0.000, B 0.000, C 0.000 }
gfCNCPoint2[26276] = {X 520.6107, Y 21.6857, Z -3.8333, A 0.000, B 0.000, C 0.000 }
gfCNCPoint2[26277] = {X 519.9691, Y 21.6857, Z -3.8333, A 0.000, B 0.000, C 0.000 }
gfCNCPoint2[26278] = {X 518.9900, Y 21.5754, Z -3.8333, A 0.000, B 0.000, C 0.000 }
gfCNCPoint2[26279] = {X 518.0600, Y 21.2500, Z -3.8333, A 0.000, B 0.000, C 0.000 }
gfCNCPoint2[26280] = {X 517.2257, Y 20.7258, Z -3.8333, A 0.000, B 0.000, C 0.000 }
gfCNCPoint2[26281] = {X 516.5290, Y 20.0291, Z -3.8333, A 0.000, B 0.000, C 0.000 }
gfCNCPoint2[26282] = {X 516.0048, Y 19.1948, Z -3.8333, A 0.000, B 0.000, C 0.000 }
gfCNCPoint2[26283] = {X 515.6794, Y 18.2648, Z -3.8333, A 0.000, B 0.000, C 0.000 }
gfCNCPoint2[26284] = {X 515.5691, Y 17.2857, Z -3.8333, A 0.000, B 0.000, C 0.000 }
gfCNCPoint2[26285] = {X 515.5691, Y 10.3077, Z -3.8333, A 0.000, B 0.000, C 0.000 }
gfCNCPoint2[26286] = {X 515.6394, Y 9.5244, Z -3.8333, A 0.000, B 0.000, C 0.000 }
gfCNCPoint2[26287] = {X 515.8480, Y 8.7662, Z -3.8333, A 0.000, B 0.000, C 0.000 }
gfCNCPoint2[26288] = {X 516.1882, Y 8.0571, Z -3.8333, A 0.000, B 0.000, C 0.000 }
gfCNCPoint2[26289] = {X 516.6493, Y 7.4200, Z -3.8333, A 0.000, B 0.000, C 0.000 }
gfCNCPoint2[26290] = {X 516.2871, Y 7.1050, Z -3.8333, A 0.000, B 0.000, C 0.000 }
gfCNCPoint2[26291] = {X 469.2607, Y 7.1050, Z -3.8333, A 0.000, B 0.000, C 0.000 }
gfCNCPoint2[26292] = {X 469.2607, Y 11.9050, Z -3.8333, A 0.000, B 0.000, C 0.000 }
gfCNCPoint2[26293] = {X 469.1140, Y 11.9050, Z -3.8333, A 0.000, B 0.000, C 0.000 }
gfCNCPoint2[26294] = {X 469.1170, Y 12.0438, Z -3.8333, A 0.000, B 0.000, C 0.000 }
gfCNCPoint2[26295] = {X 469.1179, Y 12.1827, Z -3.8333, A 0.000, B 0.000, C 0.000 }
gfCNCPoint2[26296] = {X 469.1887, Y 12.0435, Z -3.8333, A 0.000, B 0.000, C 0.000 }
gfCNCPoint2[26297] = {X 469.2607, Y 11.9050, Z -3.8333, A 0.000, B 0.000, C 0.000 }
gfCNCPoint2[26298] = {X 469.2607, Y 9.5050, Z -3.8333, A 0.000, B 0.000, C 0.000 }
gfCNCPoint2[26299] = {X 466.2072, Y 9.5050, Z -3.8333, A 0.000, B 0.000, C 0.000 }
gfCNCPoint2[26300] = {X 466.5688, Y 10.7172, Z -3.8333, A 0.000, B 0.000, C 0.000 }
gfCNCPoint2[26301] = {X 466.7150, Y 11.9738, Z -3.8333, A 0.000, B 0.000, C 0.000 }
gfCNCPoint2[26302] = {X 466.7172, Y 12.0780, Z -3.8333, A 0.000, B 0.000, C 0.000 }
gfCNCPoint2[26303] = {X 466.7179, Y 12.1822, Z -3.8333, A 0.000, B 0.000, C 0.000 }
gfCNCPoint2[26304] = {X 466.7179, Y 12.9779, Z -3.8333, A 0.000, B 0.000, C 0.000 }
gfCNCPoint2[26305] = {X 466.6191, Y 14.1735, Z -3.8333, A 0.000, B 0.000, C 0.000 }
gfCNCPoint2[26306] = {X 466.3253, Y 15.3365, Z -3.8333, A 0.000, B 0.000, C 0.000 }
gfCNCPoint2[26307] = {X 465.8445, Y 16.4356, Z -3.8333, A 0.000, B 0.000, C 0.000 }
gfCNCPoint2[26308] = {X 465.1897, Y 17.4407, Z -3.8333, A 0.000, B 0.000, C 0.000 }
gfCNCPoint2[26309] = {X 465.1901, Y 25.8743, Z -3.8333, A 0.000, B 0.000, C 0.000 }
gfCNCPoint2[26310] = {X 467.5901, Y 25.8742, Z -3.8333, A 0.000, B 0.000, C 0.000 }
gfCNCPoint2[26311] = {X 467.5907, Y 38.9900, Z -3.8333, A 0.000, B 0.000, C 0.000 }
gfCNCPoint2[26312] = {X 467.6015, Y 39.0069, Z -3.8333, A 0.000, B 0.000, C 0.000 }
gfCNCPoint2[26313] = {X 468.3506, Y 37.9855, Z -3.8333, A 0.000, B 0.000, C 0.000 }
gfCNCPoint2[26314] = {X 469.2267, Y 37.0706, Z -3.8333, A 0.000, B 0.000, C 0.000 }
gfCNCPoint2[26315] = {X 470.2148, Y 36.2780, Z -3.8333, A 0.000, B 0.000, C 0.000 }
gfCNCPoint2[26316] = {X 471.5279, Y 33.7077, Z -3.8333, A 0.000, B 0.000, C 0.000 }
gfCNCPoint2[26317] = {X 470.4808, Y 32.4115, Z -3.8333, A 0.000, B 0.000, C 0.000 }
gfCNCPoint2[26318] = {X 469.5671, Y 31.0181, Z -3.8333, A 0.000, B 0.000, C 0.000 }
gfCNCPoint2[26319] = {X 468.7956, Y 29.5411, Z -3.8333, A 0.000, B 0.000, C 0.000 }
gfCNCPoint2[26320] = {X 468.1739, Y 27.9951, Z -3.8333, A 0.000, B 0.000, C 0.000 }
gfCNCPoint2[26321] = {X 467.7082, Y 26.3952, Z -3.8333, A 0.000, B 0.000, C 0.000 }
gfCNCPoint2[26322] = {X 467.6475, Y 26.1351, Z -3.8333, A 0.000, B 0.000, C 0.000 }
gfCNCPoint2[26323] = {X 467.5901, Y 25.8742, Z -3.8333, A 0.000, B 0.000, C 0.000 }
gfCNCPoint2[26324] = {X 465.1901, Y 25.8743, Z -3.8333, A 0.000, B 0.000, C 0.000 }
gfCNCPoint2[26325] = {X 465.1907, Y 39.7474, Z -3.8333, A 0.000, B 0.000, C 0.000 }
gfCNCPoint2[26326] = {X 465.3904, Y 40.0175, Z -3.8333, A 0.000, B 0.000, C 0.000 }
gfCNCPoint2[26327] = {X 465.5774, Y 40.2966, Z -3.8333, A 0.000, B 0.000, C 0.000 }
gfCNCPoint2[26328] = {X 466.0634, Y 41.1919, Z -3.8333, A 0.000, B 0.000, C 0.000 }
gfCNCPoint2[26329] = {X 466.4196, Y 42.1462, Z -3.8333, A 0.000, B 0.000, C 0.000 }
gfCNCPoint2[26330] = {X 466.6392, Y 43.1408, Z -3.8333, A 0.000, B 0.000, C 0.000 }
gfCNCPoint2[26331] = {X 466.7178, Y 44.1564, Z -3.8333, A 0.000, B 0.000, C 0.000 }
gfCNCPoint2[26332] = {X 466.7179, Y 45.0000, Z -3.8333, A 0.000, B 0.000, C 0.000 }
gfCNCPoint2[26333] = {X 466.7033, Y 45.4609, Z -3.8333, A 0.000, B 0.000, C 0.000 }
gfCNCPoint2[26334] = {X 466.6596, Y 45.9200, Z -3.8333, A 0.000, B 0.000, C 0.000 }
gfCNCPoint2[26335] = {X 468.5433, Y 45.9200, Z -3.8333, A 0.000, B 0.000, C 0.000 }
gfCNCPoint2[26336] = {X 468.4996, Y 45.4609, Z -3.8333, A 0.000, B 0.000, C 0.000 }
gfCNCPoint2[26337] = {X 468.4850, Y 45.0000, Z -3.8333, A 0.000, B 0.000, C 0.000 }
gfCNCPoint2[26338] = {X 468.4850, Y 44.2090, Z -3.8333, A 0.000, B 0.000, C 0.000 }
gfCNCPoint2[26339] = {X 468.5580, Y 43.1798, Z -3.8333, A 0.000, B 0.000, C 0.000 }
gfCNCPoint2[26340] = {X 468.7759, Y 42.1714, Z -3.8333, A 0.000, B 0.000, C 0.000 }
gfCNCPoint2[26341] = {X 469.1341, Y 41.2038, Z -3.8333, A 0.000, B 0.000, C 0.000 }
gfCNCPoint2[26342] = {X 469.6255, Y 40.2966, Z -3.8333, A 0.000, B 0.000, C 0.000 }
gfCNCPoint2[26343] = {X 470.3102, Y 39.3876, Z -3.8333, A 0.000, B 0.000, C 0.000 }
gfCNCPoint2[26344] = {X 471.1282, Y 38.5964, Z -3.8333, A 0.000, B 0.000, C 0.000 }
gfCNCPoint2[26345] = {X 472.0595, Y 37.9424, Z -3.8333, A 0.000, B 0.000, C 0.000 }
gfCNCPoint2[26346] = {X 474.4571, Y 33.2494, Z -3.8333, A 0.000, B 0.000, C 0.000 }
gfCNCPoint2[26347] = {X 473.2256, Y 32.0046, Z -3.8333, A 0.000, B 0.000, C 0.000 }
gfCNCPoint2[26348] = {X 472.1539, Y 30.6198, Z -3.8333, A 0.000, B 0.000, C 0.000 }
gfCNCPoint2[26349] = {X 471.2578, Y 29.1155, Z -3.8333, A 0.000, B 0.000, C 0.000 }
gfCNCPoint2[26350] = {X 470.5506, Y 27.5136, Z -3.8333, A 0.000, B 0.000, C 0.000 }
gfCNCPoint2[26351] = {X 470.0426, Y 25.8379, Z -3.8333, A 0.000, B 0.000, C 0.000 }
gfCNCPoint2[26352] = {X 469.9883, Y 25.6052, Z -3.8333, A 0.000, B 0.000, C 0.000 }
gfCNCPoint2[26353] = {X 469.9369, Y 25.3719, Z -3.8333, A 0.000, B 0.000, C 0.000 }
gfCNCPoint2[26354] = {X 469.6272, Y 23.4787, Z -3.8333, A 0.000, B 0.000, C 0.000 }
gfCNCPoint2[26355] = {X 469.5028, Y 21.5644, Z -3.8333, A 0.000, B 0.000, C 0.000 }
gfCNCPoint2[26356] = {X 469.5651, Y 19.6470, Z -3.8333, A 0.000, B 0.000, C 0.000 }
gfCNCPoint2[26357] = {X 469.8134, Y 17.7448, Z -3.8333, A 0.000, B 0.000, C 0.000 }
gfCNCPoint2[26358] = {X 470.2453, Y 15.8757, Z -3.8333, A 0.000, B 0.000, C 0.000 }
gfCNCPoint2[26359] = {X 470.6916, Y 14.5441, Z -3.8333, A 0.000, B 0.000, C 0.000 }
gfCNCPoint2[26360] = {X 471.2622, Y 13.2608, Z -3.8333, A 0.000, B 0.000, C 0.000 }
gfCNCPoint2[26361] = {X 471.3230, Y 13.1410, Z -3.8333, A 0.000, B 0.000, C 0.000 }
gfCNCPoint2[26362] = {X 471.3850, Y 13.0219, Z -3.8333, A 0.000, B 0.000, C 0.000 }
gfCNCPoint2[26363] = {X 472.1261, Y 11.7667, Z -3.8333, A 0.000, B 0.000, C 0.000 }
gfCNCPoint2[26364] = {X 472.9871, Y 10.5906, Z -3.8333, A 0.000, B 0.000, C 0.000 }
gfCNCPoint2[26365] = {X 473.9597, Y 9.5050, Z -3.8333, A 0.000, B 0.000, C 0.000 }
gfCNCPoint2[26366] = {X 469.2607, Y 9.5050, Z -3.8333, A 0.000, B 0.000, C 0.000 }
gfCNCPoint2[26367] = {X 469.2607, Y 7.1050, Z -3.8333, A 0.000, B 0.000, C 0.000 }
gfCNCPoint2[26368] = {X 370.1024, Y 7.1050, Z -3.8333, A 0.000, B 0.000, C 0.000 }
gfCNCPoint2[26369] = {X 371.1260, Y 8.7919, Z -3.8333, A 0.000, B 0.000, C 0.000 }
gfCNCPoint2[26370] = {X 372.0367, Y 10.5423, Z -3.8333, A 0.000, B 0.000, C 0.000 }
gfCNCPoint2[26371] = {X 372.9295, Y 12.5982, Z -3.8333, A 0.000, B 0.000, C 0.000 }
gfCNCPoint2[26372] = {X 373.6667, Y 14.7148, Z -3.8333, A 0.000, B 0.000, C 0.000 }
gfCNCPoint2[26373] = {X 374.2442, Y 16.8804, Z -3.8333, A 0.000, B 0.000, C 0.000 }
gfCNCPoint2[26374] = {X 374.7325, Y 19.4464, Z -3.8333, A 0.000, B 0.000, C 0.000 }
gfCNCPoint2[26375] = {X 375.0383, Y 22.0405, Z -3.8333, A 0.000, B 0.000, C 0.000 }
gfCNCPoint2[26376] = {X 375.1603, Y 24.6497, Z -3.8333, A 0.000, B 0.000, C 0.000 }
gfCNCPoint2[26377] = {X 375.0978, Y 27.2610, Z -3.8333, A 0.000, B 0.000, C 0.000 }
gfCNCPoint2[26378] = {X 374.8511, Y 29.8614, Z -3.8333, A 0.000, B 0.000, C 0.000 }
gfCNCPoint2[26379] = {X 374.4214, Y 32.4379, Z -3.8333, A 0.000, B 0.000, C 0.000 }
gfCNCPoint2[26380] = {X 373.7849, Y 34.9950, Z -3.8333, A 0.000, B 0.000, C 0.000 }
gfCNCPoint2[26381] = {X 372.9255, Y 37.4860, Z -3.8333, A 0.000, B 0.000, C 0.000 }
